# B&R Automation Studio project NAELD004C00R10L518F00 (part 10)

#### Act_OptP0410Navi.st
```iecst
ACTION Act_OptP0410Navi:

	IF tyP0410MagSel.tyNavi2Lyr1.tyBtnBack.bRtCompl = TRUE
		OR tyP0410MagSel.tyNavi2Lyr2.tyBtnBack.bRtCompl = TRUE
		OR tyP0410MagSel.tyNavi1Lyr1.tyBtnBack.bRtCompl = TRUE
		THEN
		tyP0410MagSel.tyNavi2Lyr1.tyBtnBack.bRtCompl := FALSE;
		tyP0410MagSel.tyNavi2Lyr1.tyBtnBack.bValue	:= FALSE;
		tyP0410MagSel.tyNavi2Lyr2.tyBtnBack.bRtCompl := FALSE;
		tyP0410MagSel.tyNavi2Lyr2.tyBtnBack.bValue	:= FALSE;

		tyP0410MagSel.tyNavi1Lyr1.tyBtnBack.bRtCompl := FALSE;
		tyP0410MagSel.tyNavi1Lyr1.tyBtnBack.bValue := FALSE;

		eChgPage	:= UIP0002Menu;

	ELSIF tyP0410MagSel.tyNavi2Lyr1.tyBtnLeft.bRtCompl = TRUE OR tyP0410MagSel.tyNavi2Lyr1.tyBtnRgt.bRtCompl = TRUE THEN
		tyP0410MagSel.tyNavi2Lyr1.tyBtnLeft.bRtCompl	:= FALSE;
		tyP0410MagSel.tyNavi2Lyr1.tyBtnRgt.bRtCompl	:= FALSE;

		p_tyC0004Navi ACCESS ADR(tyP0410MagSel.tyNavi2Lyr2);

		bRefreshMagRcpTable := TRUE;
		bMagazineRcpA := FALSE;
		bMagazineRcpB := TRUE;

		fUIInRtStatHide(ADR(tyP0410MagSel.tyMagDet.tyLyr.uiRtStat));

		tyP0410MagSel.tyMagSel.tyTxtMagTitle.usiValueIdx := 127;

		tyP0410MagSel.tyMagSel.tyStringRecipeNm.sValue			:= p_tyMagRcpCurrRcp1.sRcpNm;
		tyP0410MagSel.tyMagSel.tyNumMaxSlt.diValue				:= p_tyMagRcpCurrRcp1.diTtlSlt;
		tyP0410MagSel.tyMagSel.tyNumSltToSltDist.diValue		:= p_tyMagRcpCurrRcp1.diSltToSltInUM;
		tyP0410MagSel.tyMagSel.tyNumLifterMag1Slt1Pos.diValue	:= p_tyMagRcpCurrRcp1.diMag1Slt1PosInUM;
		tyP0410MagSel.tyMagSel.tyNumLifterMag2Slt1Pos.diValue	:= p_tyMagRcpCurrRcp1.diMag2Slt1PosInUM;
		tyP0410MagSel.tyMagSel.tyNumLifterMag3Slt1Pos.diValue	:= p_tyMagRcpCurrRcp1.diMag3Slt1PosInUM;
		tyP0410MagSel.tyMagSel.tyNumLifterMag4Slt1Pos.diValue	:= p_tyMagRcpCurrRcp1.diMag4Slt1PosInUM;
		tyP0410MagSel.tyMagSel.tyNumTravPosMag1.diValue			:= p_tyMagRcpCurrRcp1.diMag1TravPosInUM;
		tyP0410MagSel.tyMagSel.tyNumTravPosMag2.diValue			:= p_tyMagRcpCurrRcp1.diMag2TravPosInUM;
		tyP0410MagSel.tyMagSel.tyNumTravPosMag3.diValue			:= p_tyMagRcpCurrRcp1.diMag3TravPosInUM;
		tyP0410MagSel.tyMagSel.tyNumTravPosMag4.diValue			:= p_tyMagRcpCurrRcp1.diMag4TravPosInUM;
		tyP0410MagSel.tyMagSel.tyTxtMagModel.usiValueIdx		:= p_tyMagRcpCurrRcp1.usiMagModel;
		tyP0410MagSel.tyMagSel.tyNumMagMaxBrdWidth.diValue		:= p_tyMagRcpCurrRcp1.diMagMaxBrdWidth;
		tyP0410MagSel.tyMagSel.tyBtnSafetyBar.bValue			:= p_tyMagRcpCurrRcp1.bSafetyBarDisabled;

	ELSIF tyP0410MagSel.tyNavi2Lyr2.tyBtnLeft.bRtCompl = TRUE OR tyP0410MagSel.tyNavi2Lyr2.tyBtnRgt.bRtCompl = TRUE THEN
		tyP0410MagSel.tyNavi2Lyr2.tyBtnLeft.bRtCompl	:= FALSE;
		tyP0410MagSel.tyNavi2Lyr2.tyBtnRgt.bRtCompl	:= FALSE;

		p_tyC0004Navi ACCESS ADR(tyP0410MagSel.tyNavi2Lyr1);

		bRefreshMagRcpTable := TRUE;
		bMagazineRcpA := TRUE;
		bMagazineRcpB := FALSE;

		fUIInRtStatHide(ADR(tyP0410MagSel.tyMagDet.tyLyr.uiRtStat));

		tyP0410MagSel.tyMagSel.tyTxtMagTitle.usiValueIdx := 126;

		tyP0410MagSel.tyMagSel.tyStringRecipeNm.sValue			:= p_tyMagRcpCurrRcp.sRcpNm;
		tyP0410MagSel.tyMagSel.tyNumMaxSlt.diValue				:= p_tyMagRcpCurrRcp.diTtlSlt;
		tyP0410MagSel.tyMagSel.tyNumSltToSltDist.diValue		:= p_tyMagRcpCurrRcp.diSltToSltInUM;
		tyP0410MagSel.tyMagSel.tyNumLifterMag1Slt1Pos.diValue	:= p_tyMagRcpCurrRcp.diMag1Slt1PosInUM;
		tyP0410MagSel.tyMagSel.tyNumLifterMag2Slt1Pos.diValue	:= p_tyMagRcpCurrRcp.diMag2Slt1PosInUM;
		tyP0410MagSel.tyMagSel.tyNumLifterMag3Slt1Pos.diValue	:= p_tyMagRcpCurrRcp.diMag3Slt1PosInUM;
		tyP0410MagSel.tyMagSel.tyNumLifterMag4Slt1Pos.diValue	:= p_tyMagRcpCurrRcp.diMag4Slt1PosInUM;
		tyP0410MagSel.tyMagSel.tyNumTravPosMag1.diValue			:= p_tyMagRcpCurrRcp.diMag1TravPosInUM;
		tyP0410MagSel.tyMagSel.tyNumTravPosMag2.diValue			:= p_tyMagRcpCurrRcp.diMag2TravPosInUM;
		tyP0410MagSel.tyMagSel.tyNumTravPosMag3.diValue			:= p_tyMagRcpCurrRcp.diMag3TravPosInUM;
		tyP0410MagSel.tyMagSel.tyNumTravPosMag4.diValue			:= p_tyMagRcpCurrRcp.diMag4TravPosInUM;
		tyP0410MagSel.tyMagSel.tyTxtMagModel.usiValueIdx		:= p_tyMagRcpCurrRcp.usiMagModel;
		tyP0410MagSel.tyMagSel.tyNumMagMaxBrdWidth.diValue		:= p_tyMagRcpCurrRcp.diMagMaxBrdWidth;
		tyP0410MagSel.tyMagSel.tyBtnSafetyBar.bValue			:= p_tyMagRcpCurrRcp.bSafetyBarDisabled;
	END_IF

END_ACTION
```

#### Act_OptP0410Mask.st
```iecst
ACTION Act_OptP0410Mask:

	IF tyP0410MagSel.tyMagSel.tyBtnLoad.bRtCompl = FALSE THEN
		IF tyP0410MagSel.tyMagSel.tyTableRecipe.a_tyStringDataCol1[tyP0410Table.uiSelectedRow].sValue = '' THEN
			fUIInRtStatOff(ADR(tyP0410MagSel.tyMagSel.tyBtnLoad.uiMaskRtStat));
			fUIInRtStatOff(ADR(tyP0410MagSel.tyMagSel.tyBtnPreview.uiMaskRtStat));
		ELSE
			fUIInRtStatHide(ADR(tyP0410MagSel.tyMagSel.tyBtnLoad.uiMaskRtStat));
			fUIInRtStatHide(ADR(tyP0410MagSel.tyMagSel.tyBtnPreview.uiMaskRtStat));
		END_IF
	END_IF

	tyP0410MagSel.tyMagSel.tyBtnSort.uiMaskRtStat.0		:= (tyP0410MagSel1.tyMagSel.tyTableRecipe.a_tyStringDataCol1[1].sValue <> '') AND (tyP0410MagSel1.tyMagSel.tyBtnLoad.bRtCompl = FALSE);

END_ACTION
```

#### Act_OptP0410Load.st
```iecst
ACTION Act_OptP0410Load:

	IF tyP0410MagSel.tyMagSel.tyBtnLoad.bRtCompl = TRUE THEN

		IF usiSelMagRcpStep = 0 THEN
			//Message Confirmation Ask
			//Mask
			tyP0410MagSel.tyMagSel.tyTableRecipe.uiMaskRtStat.0		:= FALSE;
			tyP0410MagSel.tyMagSel.tyBtnPreview.uiMaskRtStat.0		:= FALSE;

			p_tyC0008MsgBox ACCESS ADR(tyP0410MagSel.tyMsgBoxSelRcpAsk);

			IF tyP0410MagSel.tyMsgBoxSelRcpAsk.tyBtnYes.bRtCompl = TRUE THEN
				tyP0410MagSel.tyMsgBoxSelRcpAsk.tyBtnYes.bRtCompl	:= FALSE;
				tyP0410MagSel.tyMsgBoxSelRcpAsk.tyBtnYes.bValue		:= FALSE;

				p_tyC0008MsgBox ACCESS ADR(tyP0410MagSel.tyMsgBoxHide);

				usiSelMagRcpStep		:= 1;

			ELSIF tyP0410MagSel.tyMsgBoxSelRcpAsk.tyBtnNo.bRtCompl = TRUE THEN
				tyP0410MagSel.tyMsgBoxSelRcpAsk.tyBtnNo.bRtCompl	:= FALSE;
				tyP0410MagSel.tyMsgBoxSelRcpAsk.tyBtnNo.bValue		:= FALSE;

				p_tyC0008MsgBox ACCESS ADR(tyP0410MagSel.tyMsgBoxHide);

				usiSelMagRcpStep		:= 99;

			END_IF

		ELSIF usiSelMagRcpStep = 1 THEN
			//Load Magazine Recipe

			IF bMagazineRcpA THEN
				tyMagRcpInfoIn.sRcpNm		:= tyP0410MagSel.tyMagSel.tyTableRecipe.a_tyStringDataCol1[tyP0410Table.uiSelectedRow].sValue;

				eMagRcpAct	:= MagRcpActLoadRcp;

				IF p_eMagRcpStat = MagRcpActLoadRcp AND p_eMagRcpStatus = Done THEN
					eMagRcpAct	:= MagRcpActIdle;

					IF p_bMagRcpNmEmpty = TRUE AND p_bMagRcpNmNotExist = TRUE THEN
						usiSelMagRcpStep	:= 2;
					ELSE

							//Update UI Current Recipe
							tyP0410MagSel.tyMagSel.tyStringRecipeNm.sValue			:= p_tyMagRcpCurrRcp.sRcpNm;
							tyP0410MagSel.tyMagSel.tyNumSltToSltDist.diValue		:= p_tyMagRcpCurrRcp.diSltToSltInUM;
							tyP0410MagSel.tyMagSel.tyNumMaxSlt.diValue				:= p_tyMagRcpCurrRcp.diTtlSlt;
							tyP0410MagSel.tyMagSel.tyNumLifterMag1Slt1Pos.diValue	:= p_tyMagRcpCurrRcp.diMag1Slt1PosInUM;
							tyP0410MagSel.tyMagSel.tyNumLifterMag2Slt1Pos.diValue	:= p_tyMagRcpCurrRcp.diMag2Slt1PosInUM;
							tyP0410MagSel.tyMagSel.tyNumLifterMag3Slt1Pos.diValue	:= p_tyMagRcpCurrRcp.diMag3Slt1PosInUM;
							tyP0410MagSel.tyMagSel.tyNumLifterMag4Slt1Pos.diValue	:= p_tyMagRcpCurrRcp.diMag4Slt1PosInUM;
							tyP0410MagSel.tyMagSel.tyNumTravPosMag1.diValue			:= p_tyMagRcpCurrRcp.diMag1TravPosInUM;
							tyP0410MagSel.tyMagSel.tyNumTravPosMag2.diValue			:= p_tyMagRcpCurrRcp.diMag2TravPosInUM;
							tyP0410MagSel.tyMagSel.tyNumTravPosMag3.diValue			:= p_tyMagRcpCurrRcp.diMag3TravPosInUM;
							tyP0410MagSel.tyMagSel.tyNumTravPosMag4.diValue			:= p_tyMagRcpCurrRcp.diMag4TravPosInUM;
							tyP0410MagSel.tyMagSel.tyTxtMagModel.usiValueIdx		:= p_tyMagRcpCurrRcp.usiMagModel;
							tyP0410MagSel.tyMagSel.tyNumMagMaxBrdWidth.diValue		:= p_tyMagRcpCurrRcp.diMagMaxBrdWidth;
							tyP0410MagSel.tyMagSel.tyBtnSafetyBar.bValue			:= p_tyMagRcpCurrRcp.bSafetyBarDisabled;
							tyP0410MagSel.tyMagSel.tyBtnMagHeightChkEn.bValue		:= p_tyMagRcpCurrRcp.bMagHeightChkEn;

							tyMagRcpCurrRcpWr	:= p_tyMagRcpCurrRcp;

							usiSelMagRcpStep	:= 99;
						END_IF

					ELSIF p_eMagRcpStatus = Error THEN
						eMagRcpAct	:= MagRcpActIdle;
						usiSelMagRcpStep		:= 99;

					END_IF

				ELSIF usiSelMagRcpStep = 2 THEN
					//Message Name Not Found
					p_tyC0008MsgBox ACCESS ADR(tyP0410MagSel.tyMsgBoxSelRcpNoNm);

					IF tyP0410MagSel.tyMsgBoxSelRcpNoNm.tyBtnNo.bRtCompl = TRUE THEN
						tyP0410MagSel.tyMsgBoxSelRcpNoNm.tyBtnNo.bRtCompl	:= FALSE;
						tyP0410MagSel.tyMsgBoxSelRcpNoNm.tyBtnNo.bValue		:= FALSE;

					p_tyC0008MsgBox ACCESS ADR(tyP0410MagSel.tyMsgBoxHide);

					usiSelMagRcpStep		:= 99;

				END_IF

			ELSIF bMagazineRcpB THEN
				tyMagRcpInfoIn1.sRcpNm		:= tyP0410MagSel.tyMagSel.tyTableRecipe.a_tyStringDataCol1[tyP0410Table.uiSelectedRow].sValue;

				eMagRcpAct1	:= MagRcpActLoadRcp;

				IF p_eMagRcpStat1 = MagRcpActLoadRcp AND p_eMagRcpStatus1 = Done THEN
					eMagRcpAct1	:= MagRcpActIdle;

					IF p_bMagRcpNmEmpty1 = TRUE AND p_bMagRcpNmNotExist1 = TRUE THEN
						usiSelMagRcpStep	:= 2;
					ELSE

						//Update UI Current Recipe
						tyP0410MagSel.tyMagSel.tyStringRecipeNm.sValue			:= p_tyMagRcpCurrRcp1.sRcpNm;
						tyP0410MagSel.tyMagSel.tyNumSltToSltDist.diValue		:= p_tyMagRcpCurrRcp1.diSltToSltInUM;
						tyP0410MagSel.tyMagSel.tyNumMaxSlt.diValue				:= p_tyMagRcpCurrRcp1.diTtlSlt;
						tyP0410MagSel.tyMagSel.tyNumLifterMag1Slt1Pos.diValue	:= p_tyMagRcpCurrRcp1.diMag1Slt1PosInUM;
						tyP0410MagSel.tyMagSel.tyNumLifterMag2Slt1Pos.diValue	:= p_tyMagRcpCurrRcp1.diMag2Slt1PosInUM;
						tyP0410MagSel.tyMagSel.tyNumLifterMag3Slt1Pos.diValue	:= p_tyMagRcpCurrRcp1.diMag3Slt1PosInUM;
						tyP0410MagSel.tyMagSel.tyNumLifterMag4Slt1Pos.diValue	:= p_tyMagRcpCurrRcp1.diMag4Slt1PosInUM;
						tyP0410MagSel.tyMagSel.tyNumTravPosMag1.diValue			:= p_tyMagRcpCurrRcp1.diMag1TravPosInUM;
						tyP0410MagSel.tyMagSel.tyNumTravPosMag2.diValue			:= p_tyMagRcpCurrRcp1.diMag2TravPosInUM;
						tyP0410MagSel.tyMagSel.tyNumTravPosMag3.diValue			:= p_tyMagRcpCurrRcp1.diMag3TravPosInUM;
						tyP0410MagSel.tyMagSel.tyNumTravPosMag4.diValue			:= p_tyMagRcpCurrRcp1.diMag4TravPosInUM;
						tyP0410MagSel.tyMagSel.tyTxtMagModel.usiValueIdx		:= p_tyMagRcpCurrRcp1.usiMagModel;
						tyP0410MagSel.tyMagSel.tyNumMagMaxBrdWidth.diValue		:= p_tyMagRcpCurrRcp1.diMagMaxBrdWidth;
						tyP0410MagSel.tyMagSel.tyBtnSafetyBar.bValue			:= p_tyMagRcpCurrRcp1.bSafetyBarDisabled;
						tyP0410MagSel.tyMagSel.tyBtnMagHeightChkEn.bValue		:= p_tyMagRcpCurrRcp1.bMagHeightChkEn;

						tyMagRcpCurrRcpWr1	:= p_tyMagRcpCurrRcp1;

						usiSelMagRcpStep	:= 99;
					END_IF

				ELSIF p_eMagRcpStatus = Error THEN
					eMagRcpAct1	:= MagRcpActIdle;
					usiSelMagRcpStep		:= 99;

				END_IF

			ELSIF usiSelMagRcpStep = 2 THEN
				//Message Name Not Found
				p_tyC0008MsgBox ACCESS ADR(tyP0410MagSel.tyMsgBoxSelRcpNoNm);

				IF tyP0410MagSel.tyMsgBoxSelRcpNoNm.tyBtnNo.bRtCompl = TRUE THEN
					tyP0410MagSel.tyMsgBoxSelRcpNoNm.tyBtnNo.bRtCompl	:= FALSE;
					tyP0410MagSel.tyMsgBoxSelRcpNoNm.tyBtnNo.bValue		:= FALSE;

					p_tyC0008MsgBox ACCESS ADR(tyP0410MagSel.tyMsgBoxHide);

					usiSelMagRcpStep		:= 99;

				END_IF
			END_IF

		ELSIF usiSelMagRcpStep = 99 THEN
			//Complete
			//Unmask
			tyP0410MagSel.tyMagSel.tyTableRecipe.uiMaskRtStat.0		:= TRUE;
			tyP0410MagSel.tyMagSel.tyBtnPreview.uiMaskRtStat.0		:= TRUE;

			//Reset
			tyP0410MagSel.tyMagSel.tyBtnLoad.bRtCompl				:= FALSE;
			tyP0410MagSel.tyMagSel.tyBtnLoad.bValue					:= FALSE;

			usiSelMagRcpStep			:= 0;

		END_IF

	END_IF

END_ACTION
```

#### Act_OptP0410Preview.st
```iecst
ACTION Act_OptP0410Preview:

	IF tyP0410MagSel.tyMagSel.tyBtnPreview.bRtCompl = TRUE THEN
		IF bMagazineRcpA THEN
			tyMagRcpInfoIn.sRcpNm	:= tyP0410MagSel.tyMagSel.tyTableRecipe.a_tyStringDataCol1[tyP0410Table.uiSelectedRow].sValue;

			eMagRcpAct				:= MagRcpActGetInfo;

			IF	p_eMagRcpStat = MagRcpActGetInfo AND p_eMagRcpStatus = Done THEN
				eMagRcpAct			:= MagRcpActIdle;

				IF p_bMagRcpNmEmpty = TRUE AND p_bMagRcpNmNotExist = TRUE THEN

					tyP0410MagSel.tyMagDet.tyStringRecipeNm.sValue			:= '';
					tyP0410MagSel.tyMagDet.tyNumSltToSltDist.diValue		:= 0;
					tyP0410MagSel.tyMagDet.tyNumMaxSlt.diValue				:= 0;
					tyP0410MagSel.tyMagDet.tyNumLifterMag1Slt1Pos.diValue	:= 0;
					tyP0410MagSel.tyMagDet.tyNumLifterMag2Slt1Pos.diValue	:= 0;
					tyP0410MagSel.tyMagDet.tyNumLifterMag3Slt1Pos.diValue	:= 0;
					tyP0410MagSel.tyMagDet.tyNumLifterMag4Slt1Pos.diValue	:= 0;
					tyP0410MagSel.tyMagDet.tyNumTravPosMag1.diValue			:= 0;
					tyP0410MagSel.tyMagDet.tyNumTravPosMag2.diValue			:= 0;
					tyP0410MagSel.tyMagDet.tyNumTravPosMag3.diValue			:= 0;
					tyP0410MagSel.tyMagDet.tyNumTravPosMag4.diValue			:= 0;
					tyP0410MagSel.tyMagDet.tyNumMagMaxBrdWidth.diValue		:= 0;
					tyP0410MagSel.tyMagDet.tyBtnSafetyBar.bValue			:= FALSE;
					tyP0410MagSel.tyMagDet.tyBtnMagHeightChkEn.bValue		:= FALSE;

				ELSE

					tyP0410MagSel.tyMagDet.tyStringRecipeNm.sValue			:= p_tyMagRcpInfoOut.sRcpNm;
					tyP0410MagSel.tyMagDet.tyNumSltToSltDist.diValue		:= p_tyMagRcpInfoOut.diSltToSltInUM;
					tyP0410MagSel.tyMagDet.tyNumMaxSlt.diValue				:= p_tyMagRcpInfoOut.diTtlSlt;
					tyP0410MagSel.tyMagDet.tyNumLifterMag1Slt1Pos.diValue	:= p_tyMagRcpInfoOut.diMag1Slt1PosInUM;
					tyP0410MagSel.tyMagDet.tyNumLifterMag2Slt1Pos.diValue	:= p_tyMagRcpInfoOut.diMag2Slt1PosInUM;
					tyP0410MagSel.tyMagDet.tyNumLifterMag3Slt1Pos.diValue	:= p_tyMagRcpInfoOut.diMag3Slt1PosInUM;
					tyP0410MagSel.tyMagDet.tyNumLifterMag4Slt1Pos.diValue	:= p_tyMagRcpInfoOut.diMag4Slt1PosInUM;
					tyP0410MagSel.tyMagDet.tyNumTravPosMag1.diValue			:= p_tyMagRcpInfoOut.diMag1TravPosInUM;
					tyP0410MagSel.tyMagDet.tyNumTravPosMag2.diValue			:= p_tyMagRcpInfoOut.diMag2TravPosInUM;
					tyP0410MagSel.tyMagDet.tyNumTravPosMag3.diValue			:= p_tyMagRcpInfoOut.diMag3TravPosInUM;
					tyP0410MagSel.tyMagDet.tyNumTravPosMag4.diValue			:= p_tyMagRcpInfoOut.diMag4TravPosInUM;
					tyP0410MagSel.tyMagDet.tyNumMagMaxBrdWidth.diValue		:= p_tyMagRcpInfoOut.diMagMaxBrdWidth;
					tyP0410MagSel.tyMagDet.tyBtnSafetyBar.bValue			:= p_tyMagRcpInfoOut.bSafetyBarDisabled;
					tyP0410MagSel.tyMagDet.tyBtnMagHeightChkEn.bValue		:= p_tyMagRcpInfoOut.bMagHeightChkEn;
				END_IF

				fUIInRtStatOff(ADR(tyP0410MagSel.tyMagDet.tyLyr.uiRtStat));

				tyP0410MagSel.tyMagSel.tyBtnPreview.bRtCompl				:= FALSE;
			END_IF

		ELSIF bMagazineRcpB THEN

			tyMagRcpInfoIn1.sRcpNm	:= tyP0410MagSel.tyMagSel.tyTableRecipe.a_tyStringDataCol1[tyP0410Table.uiSelectedRow].sValue;

			eMagRcpAct1				:= MagRcpActGetInfo;

			IF	p_eMagRcpStat1 = MagRcpActGetInfo AND p_eMagRcpStatus1 = Done THEN
				eMagRcpAct1			:= MagRcpActIdle;

				IF p_bMagRcpNmEmpty1 = TRUE AND p_bMagRcpNmNotExist1 = TRUE THEN

					tyP0410MagSel.tyMagDet.tyStringRecipeNm.sValue			:= '';
					tyP0410MagSel.tyMagDet.tyNumSltToSltDist.diValue		:= 0;
					tyP0410MagSel.tyMagDet.tyNumMaxSlt.diValue				:= 0;
					tyP0410MagSel.tyMagDet.tyNumLifterMag1Slt1Pos.diValue	:= 0;
					tyP0410MagSel.tyMagDet.tyNumLifterMag2Slt1Pos.diValue	:= 0;
					tyP0410MagSel.tyMagDet.tyNumLifterMag3Slt1Pos.diValue	:= 0;
					tyP0410MagSel.tyMagDet.tyNumLifterMag4Slt1Pos.diValue	:= 0;
					tyP0410MagSel.tyMagDet.tyNumTravPosMag1.diValue			:= 0;
					tyP0410MagSel.tyMagDet.tyNumTravPosMag2.diValue			:= 0;
					tyP0410MagSel.tyMagDet.tyNumTravPosMag3.diValue			:= 0;
					tyP0410MagSel.tyMagDet.tyNumTravPosMag4.diValue			:= 0;
					tyP0410MagSel.tyMagDet.tyNumMagMaxBrdWidth.diValue		:= 0;
					tyP0410MagSel.tyMagDet.tyBtnSafetyBar.bValue			:= FALSE;
					tyP0410MagSel.tyMagDet.tyBtnMagHeightChkEn.bValue		:= FALSE;
				ELSE

					tyP0410MagSel.tyMagDet.tyStringRecipeNm.sValue			:= p_tyMagRcpInfoOut1.sRcpNm;
					tyP0410MagSel.tyMagDet.tyNumSltToSltDist.diValue		:= p_tyMagRcpInfoOut1.diSltToSltInUM;
					tyP0410MagSel.tyMagDet.tyNumMaxSlt.diValue				:= p_tyMagRcpInfoOut1.diTtlSlt;
					tyP0410MagSel.tyMagDet.tyNumLifterMag1Slt1Pos.diValue	:= p_tyMagRcpInfoOut1.diMag1Slt1PosInUM;
					tyP0410MagSel.tyMagDet.tyNumLifterMag2Slt1Pos.diValue	:= p_tyMagRcpInfoOut1.diMag2Slt1PosInUM;
					tyP0410MagSel.tyMagDet.tyNumLifterMag3Slt1Pos.diValue	:= p_tyMagRcpInfoOut1.diMag3Slt1PosInUM;
					tyP0410MagSel.tyMagDet.tyNumLifterMag4Slt1Pos.diValue	:= p_tyMagRcpInfoOut1.diMag4Slt1PosInUM;
					tyP0410MagSel.tyMagDet.tyNumTravPosMag1.diValue			:= p_tyMagRcpInfoOut1.diMag1TravPosInUM;
					tyP0410MagSel.tyMagDet.tyNumTravPosMag2.diValue			:= p_tyMagRcpInfoOut1.diMag2TravPosInUM;
					tyP0410MagSel.tyMagDet.tyNumTravPosMag3.diValue			:= p_tyMagRcpInfoOut1.diMag3TravPosInUM;
					tyP0410MagSel.tyMagDet.tyNumTravPosMag4.diValue			:= p_tyMagRcpInfoOut1.diMag4TravPosInUM;
					tyP0410MagSel.tyMagDet.tyNumMagMaxBrdWidth.diValue		:= p_tyMagRcpInfoOut1.diMagMaxBrdWidth;
					tyP0410MagSel.tyMagDet.tyBtnSafetyBar.bValue			:= p_tyMagRcpInfoOut1.bSafetyBarDisabled;
					tyP0410MagSel.tyMagDet.tyBtnMagHeightChkEn.bValue		:= p_tyMagRcpInfoOut1.bMagHeightChkEn;
				END_IF

				fUIInRtStatOff(ADR(tyP0410MagSel.tyMagDet.tyLyr.uiRtStat));

				tyP0410MagSel.tyMagSel.tyBtnPreview.bRtCompl				:= FALSE;
			END_IF
		END_IF
	END_IF

	IF tyP0410MagSel.tyMagDet.tyHotspotClose.bRtCompl = TRUE THEN
		tyP0410MagSel.tyMagDet.tyHotspotClose.bRtCompl					:= FALSE;
		tyP0410MagSel.tyMagSel.tyBtnPreview.bValue						:= FALSE;

		//Hide Recipe Details
		fUIInRtStatHide(ADR(tyP0410MagSel.tyMagDet.tyLyr.uiRtStat));
	END_IF

END_ACTION
```

#### Act_OptP0410Table.st
```iecst
ACTION Act_OptP0410Table:

	//Call Table FB
	fbP0410Table.sVisuNm			:= tyP0410Table.sVisuNm;
	fbP0410Table.udiWorkAreaStartX	:= 349;
	fbP0410Table.udiWorkAreaEndX	:= 768;
	fbP0410Table.udiWorkAreaStartY	:= 107;
	fbP0410Table.udiWorkAreaEndY	:= 428;
	fbP0410Table.udiMinXDist		:= 20;
	fbP0410Table.udiMinYDist		:= 20;
	fbP0410Table.uiSlideScale		:= c_uiP0410TableSize;
	fbP0410Table.iTotalData			:= UDINT_TO_INT(c_udiMagRcpMax);;
	fbP0410Table.iTotalRow			:= c_uiP0410TableSize;
	fbP0410Table(uiSliderStatus := tyP0410MagSel.tyMagSel.tyTableRecipe.tyUISlider.uiRtStat , a_tyUIHotspot := tyP0410MagSel.tyMagSel.tyTableRecipe.a_tyHotspot , uiTablePos := tyP0410Table.uiTablePos , iSliderPos := tyP0410MagSel.tyMagSel.tyTableRecipe.tyUISlider.iValue);

	tyP0410Table.uiSelectedRow		:= fbP0410Table.uiSelectedRow;
	tyP0410Table.bTableActive		:= fbP0410Table.bTableActive;
	tyP0410Table.bSliderActive		:= fbP0410Table.bSliderActive;

	//Table Content
	IF tyP0410Table.bTableActive = TRUE OR tyP0410Table.bSliderActive = TRUE OR bRefreshMagRcpTable OR bUpdateP0410Table THEN

		IF bMagazineRcpA THEN
			FOR i := 1 TO c_uiP0410TableSize DO

				IF tyP0410MagSel.tyMagSel.tyBtnSort.bValue THEN

					tyP0410MagSel.tyMagSel.tyTableRecipe.a_tyStringDataCol0[i].sValue	:= UINT_TO_STRING(tyP0410Table.uiTablePos + i - 1);
					tyP0410MagSel.tyMagSel.tyTableRecipe.a_tyStringDataCol1[i].sValue	:= p_tyMagRcpSortedList[tyP0410Table.uiTablePos + i - 1].sRcpNm;
					tyP0410MagSel.tyMagSel.tyTableRecipe.a_tyStringDataCol2[i].sValue	:= p_tyMagRcpSortedList[tyP0410Table.uiTablePos + i - 1].sDisplayInfo;

				ELSE
					tyP0410MagSel.tyMagSel.tyTableRecipe.a_tyStringDataCol0[i].sValue	    := UINT_TO_STRING(tyP0410Table.uiTablePos + i - 1);
					tyP0410MagSel.tyMagSel.tyTableRecipe.a_tyStringDataCol1[i].sValue		:= p_tyMagRcpCurrList[tyP0410Table.uiTablePos + i - 1].sRcpNm;
					tyP0410MagSel.tyMagSel.tyTableRecipe.a_tyStringDataCol2[i].sValue		:= p_tyMagRcpCurrList[tyP0410Table.uiTablePos + i - 1].sDisplayInfo;
				END_IF

			END_FOR

		ELSIF bMagazineRcpB THEN
			FOR i := 1 TO c_uiP0410TableSize DO

				IF tyP0410MagSel.tyMagSel.tyBtnSort.bValue THEN

					tyP0410MagSel.tyMagSel.tyTableRecipe.a_tyStringDataCol0[i].sValue	:= UINT_TO_STRING(tyP0410Table.uiTablePos + i - 1);
					tyP0410MagSel.tyMagSel.tyTableRecipe.a_tyStringDataCol1[i].sValue	:= p_tyMagRcpSortedList1[tyP0410Table.uiTablePos + i - 1].sRcpNm;
					tyP0410MagSel.tyMagSel.tyTableRecipe.a_tyStringDataCol2[i].sValue	:= p_tyMagRcpSortedList1[tyP0410Table.uiTablePos + i - 1].sDisplayInfo;

				ELSE
					tyP0410MagSel.tyMagSel.tyTableRecipe.a_tyStringDataCol0[i].sValue	    := UINT_TO_STRING(tyP0410Table.uiTablePos + i - 1);
					tyP0410MagSel.tyMagSel.tyTableRecipe.a_tyStringDataCol1[i].sValue		:= p_tyMagRcpCurrList1[tyP0410Table.uiTablePos + i - 1].sRcpNm;
					tyP0410MagSel.tyMagSel.tyTableRecipe.a_tyStringDataCol2[i].sValue		:= p_tyMagRcpCurrList1[tyP0410Table.uiTablePos + i - 1].sDisplayInfo;
				END_IF

			END_FOR
		END_IF

		IF bUpdateP0410Table THEN
			bUpdateP0410Table := FALSE;
		END_IF
	END_IF

	//Selected Row
	IF tyP0410Table.uiSelectedRow <> tyP0410Table.uiSelectedRowOld THEN
		FOR i := 1 TO c_uiP0410TableSize DO
			IF tyP0410Table.uiSelectedRow = i THEN
				tyP0410MagSel.tyMagSel.tyTableRecipe.a_tyStringDataCol1[i].usiColor	:= 1;
				tyP0410MagSel.tyMagSel.tyTableRecipe.a_tyStringDataCol2[i].usiColor	:= 1;
			ELSE
				tyP0410MagSel.tyMagSel.tyTableRecipe.a_tyStringDataCol1[i].usiColor	:= 0;
				tyP0410MagSel.tyMagSel.tyTableRecipe.a_tyStringDataCol2[i].usiColor	:= 0;
			END_IF

			//Magazine B
			IF tyP0410Table.uiSelectedRow = i THEN
				tyP0410MagSel1.tyMagSel.tyTableRecipe.a_tyStringDataCol1[i].usiColor	:= 1;
				tyP0410MagSel1.tyMagSel.tyTableRecipe.a_tyStringDataCol2[i].usiColor	:= 1;
			ELSE
				tyP0410MagSel1.tyMagSel.tyTableRecipe.a_tyStringDataCol1[i].usiColor	:= 0;
				tyP0410MagSel1.tyMagSel.tyTableRecipe.a_tyStringDataCol2[i].usiColor	:= 0;
			END_IF
		END_FOR

		tyP0410Table.uiSelectedRowOld	:= tyP0410Table.uiSelectedRow;
	END_IF

END_ACTION
```

#### Act_OptP0410Sort.st
```iecst
ACTION Act_OptP0410Sort:

	IF tyP0410MagSel.tyMagSel.tyBtnSort.bValue THEN
		tyP0410MagSel.tyMagSel.tyBtnSort.usiTxtIdx 	:= 1;
	ELSE
		tyP0410MagSel.tyMagSel.tyBtnSort.usiTxtIdx 	:= 0;
	END_IF

	IF tyP0410MagSel.tyMagSel.tyBtnSort.bRtCompl THEN

		IF tyP0410MagSel.tyMagSel.tyBtnSort.bValue THEN

			tyP0410MagSel.tyMagSel.tyTableRecipe.uiMaskRtStat.0	:= FALSE;

			eMagRcpAct	:= MagRcpActSort;
			eMagRcpAct1	:= MagRcpActSort;
			IF p_eMagRcpStat = MagRcpActSort AND p_eMagRcpStatus = Done
				AND (p_eMagRcpStat1 = MagRcpActSort AND p_eMagRcpStatus1 = Done)
				THEN
				eMagRcpAct		:= MagRcpActIdle;
				eMagRcpAct1		:= MagRcpActIdle;
				FOR i := 1 TO c_uiP0410TableSize DO
					tyP0410MagSel.tyMagSel.tyTableRecipe.a_tyStringDataCol0[i].sValue	:= UINT_TO_STRING(tyP0400Table.uiTablePos + i - 1);
					tyP0410MagSel.tyMagSel.tyTableRecipe.a_tyStringDataCol1[i].sValue	:= p_tyMagRcpSortedList[tyP0400Table.uiTablePos + i - 1].sRcpNm;
					tyP0410MagSel.tyMagSel.tyTableRecipe.a_tyStringDataCol2[i].sValue	:= p_tyMagRcpSortedList[tyP0400Table.uiTablePos + i - 1].sDisplayInfo;
				END_FOR

				//Unmask
				tyP0410MagSel.tyMagSel.tyTableRecipe.uiMaskRtStat.0	:= TRUE;

				tyP0410MagSel.tyMagSel.tyBtnSort.bRtCompl := FALSE;

			ELSIF p_eMagRcpStatus = Error OR p_eMagRcpStatus1 = Error THEN
				FOR i := 1 TO c_uiP0410TableSize DO
					tyP0410MagSel.tyMagSel.tyTableRecipe.a_tyStringDataCol0[i].sValue		:= UINT_TO_STRING(tyP0410Table.uiTablePos + i - 1);
					tyP0410MagSel.tyMagSel.tyTableRecipe.a_tyStringDataCol1[i].sValue		:= '';
					tyP0410MagSel.tyMagSel.tyTableRecipe.a_tyStringDataCol2[i].sValue		:= '';
				END_FOR
				eMagRcpAct		:= MagRcpActIdle;
				eMagRcpAct1		:= MagRcpActIdle;
				p_tyC0008MsgBox ACCESS ADR (tyP0410MagSel.tyMsgBoxListErr);

				IF tyP0410MagSel.tyMsgBoxListErr.tyBtnNo.bRtCompl = TRUE THEN
					tyP0410MagSel.tyMsgBoxListErr.tyBtnNo.bRtCompl 		:= TRUE;
					tyP0410MagSel.tyMsgBoxListErr.tyBtnNo.bValue			:= TRUE;

					p_tyC0008MsgBox ACCESS ADR (tyP0410MagSel.tyMsgBoxHide);

					//Unmask
					tyP0410MagSel.tyMagSel.tyTableRecipe.uiMaskRtStat.0	:= TRUE;

					//Reset
					tyP0410MagSel.tyMagSel.tyBtnSort.bRtCompl := FALSE;
				END_IF
			END_IF

		ELSE

			bUpdateP0410Table	:= TRUE;

			tyP0410MagSel.tyMagSel.tyBtnSort.bRtCompl := FALSE;

		END_IF

	END_IF

END_ACTION
```

#### Act_EntP0600Disp.st
```iecst
ACTION Act_EntP0600Disp:

	//Access Addres
	p_tyC0005Main ACCESS ADR(tyCommon.tyMain);

	p_tyC0007Notif ACCESS ADR(tyCommon.tyNotif);

	p_tyC0008MsgBox ACCESS ADR(tyP0600Alm.tyMsgBoxHide);

	p_tyC0009Info ACCESS ADR(tyCommon.tyInfo);

	p_tyC0010RcyMsg ACCESS ADR(tyP0600Alm.tyRcyMsgHide);

	p_tyP0600Alm ACCESS ADR(tyP0600Alm.tyAlm);

	tyP0600Alm.tyAlm.tyBtnCurr.bRtCompl := TRUE; //Default will be Current Alarm View

	//Reset
	bTeachTravPosA			:= FALSE;
	bTeachTravPosB			:= FALSE;
	bTeachLifterPosA		:= FALSE;
	bTeachLifterPosB		:= FALSE;
	bTeachLifterMag1Slt1Pos	:= FALSE;
	bTeachLifterMag2Slt1Pos	:= FALSE;
	bTeachLifterMag3Slt1Pos	:= FALSE;
	bTeachLifterMag4Slt1Pos	:= FALSE;
	bTeachTravPosMag1		:= FALSE;
	bTeachTravPosMag2		:= FALSE;
	bTeachTravPosMag3		:= FALSE;
	bTeachTravPosMag4		:= FALSE;
	bTeachServo				:= FALSE;

END_ACTION
```

#### Act_OptP0600Alm.st
```iecst
ACTION Act_OptP0600Alm:

	IF tyP0600Alm.tyAlm.tyBtnHistory.bRtCompl = TRUE THEN
		tyP0600Alm.tyAlm.tyBtnHistory.bRtCompl		:= FALSE;
		tyP0600Alm.tyAlm.tyBtnHistory.bValue		:= TRUE;
		tyP0600Alm.tyAlm.tyBtnCurr.bValue			:= FALSE;
	ELSIF tyP0600Alm.tyAlm.tyBtnCurr.bRtCompl = TRUE THEN
		tyP0600Alm.tyAlm.tyBtnCurr.bRtCompl			:= FALSE;
		tyP0600Alm.tyAlm.tyBtnCurr.bValue			:= TRUE;
		tyP0600Alm.tyAlm.tyBtnHistory.bValue		:= FALSE;
	END_IF

	IF NOT p_bAlarmErr THEN
		memset(ADR(tyUIAlmData.bAlm) , 0 , SIZEOF(tyUIAlmData.bAlm));
	END_IF

	IF NOT p_bAlarmWarning THEN
		memset(ADR(tyUIAlmData.bWarning) , 0 , SIZEOF(tyUIAlmData.bWarning));
	ELSE
		IF p_bDSHermesAConnected OR p_tyMcParamCurr.eDSCommA = McSetCommModSMEMA THEN
			tyUIAlmData.bWarning[3363] := FALSE;
		END_IF
		IF p_bDSHermesBConnected OR p_tyMcParamCurr.eDSCommB = McSetCommModSMEMA THEN
			tyUIAlmData.bWarning[3531] := FALSE;
		END_IF
	END_IF

	IF tyP0600Alm.tyAlm.tyBtnCurr.bValue = TRUE THEN

		fUIInRtStatOff(ADR(tyP0600Alm.tyAlm.tyAlarm.tyUIAlmCur.uiRtStat));
		fUIInRtStatHide(ADR(tyP0600Alm.tyAlm.tyAlarm.tyUIAlmHis.uiRtStat));
		tyP0600Alm.tyAlm.tyBtnHistoryUp.uiMaskRtStat.0 		:= FALSE;
		tyP0600Alm.tyAlm.tyBtnHistoryDown.uiMaskRtStat.0 	:= FALSE;

		FOR i := 1 TO c_uiP0600TableSize DO
			IF p_bStartupUISettingsLoadDone THEN
				IF p_tyAlarmCurrList[i].eSeverity = AlmSeverityError THEN
					tyUIAlmData.bAlm[p_tyAlarmCurrList[i].udiErrorCode] := p_tyAlarmCurrList[i].bAlm;
				ELSIF p_tyAlarmCurrList[i].eSeverity = AlmSeverityWarning THEN
					tyUIAlmData.bWarning[p_tyAlarmCurrList[i].udiErrorCode] := p_tyAlarmCurrList[i].bWarning;
				END_IF
			END_IF
		END_FOR

	ELSIF tyP0600Alm.tyAlm.tyBtnHistory.bValue = TRUE THEN

		fUIInRtStatHide(ADR(tyP0600Alm.tyAlm.tyAlarm.tyUIAlmCur.uiRtStat));
		fUIInRtStatOff(ADR(tyP0600Alm.tyAlm.tyAlarm.tyUIAlmHis.uiRtStat));
		tyP0600Alm.tyAlm.tyBtnHistoryUp.uiMaskRtStat.0 		:= TRUE;
		tyP0600Alm.tyAlm.tyBtnHistoryDown.uiMaskRtStat.0 	:= TRUE;

	END_IF

END_ACTION
```

#### Act_OptP0700Table.st
```iecst
ACTION Act_OptP0700Table:

	//Call Table FB
	fbP0700Table.sVisuNm			:= tyP0700Table.sVisuNm;
	fbP0700Table.udiWorkAreaStartX	:= 17;
	fbP0700Table.udiWorkAreaEndX	:= 594;
	fbP0700Table.udiWorkAreaStartY	:= 94;
	fbP0700Table.udiWorkAreaEndY	:= 445;
	fbP0700Table.udiMinXDist		:= 20;
	fbP0700Table.udiMinYDist		:= 20;
	fbP0700Table.uiSlideScale		:= c_uiP0700TableSize;
	fbP0700Table.iTotalData			:= UDINT_TO_INT(c_diLFClntNum);
	fbP0700Table.iTotalRow			:= c_uiP0700TableSize;
	fbP0700Table(uiSliderStatus 	:= tyP0700LFCtrl.tyLdr.tyTable1List.tyUISlider.uiRtStat , a_tyUIHotspot := tyP0700LFCtrl.tyLdr.tyTable1List.a_tyHotspot , uiTablePos := tyP0700Table.uiTablePos , iSliderPos := tyP0700LFCtrl.tyLdr.tyTable1List.tyUISlider.iValue);

	tyP0700Table.uiSelectedRow		:= fbP0700Table.uiSelectedRow;
	tyP0700Table.bTableActive		:= fbP0700Table.bTableActive;
	tyP0700Table.bSliderActive		:= fbP0700Table.bSliderActive;

	//Table Content
	IF tyP0700Table.bTableActive = TRUE OR tyP0700Table.bSliderActive = TRUE THEN
		FOR i := 1 TO c_uiP0700TableSize DO
			tyP0700LFCtrl.tyLdr.tyTable1List.a_tyStringDataCol0[i].sValue	:= UINT_TO_STRING(tyP0700Table.uiTablePos + i - 1);
		END_FOR
	END_IF

	//Update Status & Current Recipe
	FOR i := 1 TO c_uiP0700TableSize DO
		tyP0700LFCtrl.tyLdr.tyTable1List.a_tyStringDataCol1[i].sValue	:= p_tyLFLeaderFollowerToLeaderTag[tyP0700Table.uiTablePos + i - 1].sMcNm;
		tyP0700LFCtrl.tyLdr.tyTable1List.a_tyStringDataCol2[i].sValue	:= p_tyMcParamCurr.a_sLFIPAddr[tyP0700Table.uiTablePos + i - 1];
		tyP0700LFCtrl.tyLdr.tyTable1List.a_tyStringDataCol4[i].sValue	:= p_tyLFLeaderFollowerToLeaderTag[tyP0700Table.uiTablePos + i - 1].sCurrProdRcp;

		IF p_tyMcParamCurr.a_sLFIPAddr[tyP0700Table.uiTablePos + i - 1] = '' THEN
			tyP0700LFCtrl.tyLdr.tyTable1List.a_tyTxtDataCol3[i].usiValueIdx	:= 0;	//Empty
		ELSIF p_tyMcParamCurr.a_sLFIPAddr[tyP0700Table.uiTablePos + i - 1] = '0000' THEN
			tyP0700LFCtrl.tyLdr.tyTable1List.a_tyTxtDataCol3[i].usiValueIdx	:= 3;	//Third Party
		ELSIF p_tyMcParamCurr.a_bLFOnline[tyP0700Table.uiTablePos + i - 1] = FALSE THEN
			tyP0700LFCtrl.tyLdr.tyTable1List.a_tyTxtDataCol3[i].usiValueIdx	:= 9;	//Offline
		ELSIF p_tyMcParamCurr.a_sLFIPAddr[tyP0700Table.uiTablePos + i - 1] = p_sHWInfoIPAddr THEN
			tyP0700LFCtrl.tyLdr.tyTable1List.a_tyTxtDataCol3[i].usiValueIdx	:= 4;	//Leader
		ELSIF p_tyLFLeaderFollowerToLeaderTag[tyP0700Table.uiTablePos + i - 1].bSectionLeader = TRUE THEN
			tyP0700LFCtrl.tyLdr.tyTable1List.a_tyTxtDataCol3[i].usiValueIdx	:= 5;	//Section Leader
		ELSIF p_tyLFLeaderFollowerInfo[tyP0700Table.uiTablePos + i - 1].bOnline = FALSE THEN
			tyP0700LFCtrl.tyLdr.tyTable1List.a_tyTxtDataCol3[i].usiValueIdx	:= 9;	//Offline
		ELSE
			IF p_tyLFLeaderFollowerToLeaderTag[tyP0700Table.uiTablePos + i - 1].eCurrMachineStat=Run THEN
				IF p_tyLFLeaderFollowerToLeaderTag[tyP0700Table.uiTablePos + i - 1].eCurrMachineStat=Warning THEN
					tyP0700LFCtrl.tyLdr.tyTable1List.a_tyTxtDataCol3[i].usiValueIdx	:= 2;	//Warning
				ELSE
					tyP0700LFCtrl.tyLdr.tyTable1List.a_tyTxtDataCol3[i].usiValueIdx	:= 6;	//Run
				END_IF
			ELSE
				IF p_tyLFLeaderFollowerToLeaderTag[tyP0700Table.uiTablePos + i - 1].eCurrMachineStat=InError THEN
					tyP0700LFCtrl.tyLdr.tyTable1List.a_tyTxtDataCol3[i].usiValueIdx	:= 1;	//Error
				ELSIF p_tyLFLeaderFollowerToLeaderTag[tyP0700Table.uiTablePos + i - 1].eCurrMachineStat=Warning THEN
					tyP0700LFCtrl.tyLdr.tyTable1List.a_tyTxtDataCol3[i].usiValueIdx	:= 2;	//Warning
				ELSIF p_tyLFLeaderFollowerToLeaderTag[tyP0700Table.uiTablePos + i - 1].eCurrMachineStat=Manual THEN
					tyP0700LFCtrl.tyLdr.tyTable1List.a_tyTxtDataCol3[i].usiValueIdx	:= 8;	//Manual
				ELSE
					tyP0700LFCtrl.tyLdr.tyTable1List.a_tyTxtDataCol3[i].usiValueIdx	:= 7;	//Stop
				END_IF
			END_IF
		END_IF
	END_FOR

	//Update Color
	FOR i := 1 TO c_uiP0700TableSize DO

		IF p_tyMcParamCurr.a_sLFIPAddr[tyP0700Table.uiTablePos + i - 1] = '' THEN
			tyP0700LFCtrl.tyLdr.tyTable1List.a_tyTxtDataCol3[i].usiColor	:= 0;	//Empty
		ELSIF p_tyMcParamCurr.a_sLFIPAddr[tyP0700Table.uiTablePos + i - 1] = '0000' THEN
			tyP0700LFCtrl.tyLdr.tyTable1List.a_tyTxtDataCol3[i].usiColor	:= 0;	//Third Party
		ELSIF p_tyMcParamCurr.a_bLFOnline[tyP0700Table.uiTablePos + i - 1] = FALSE THEN
			tyP0700LFCtrl.tyLdr.tyTable1List.a_tyTxtDataCol3[i].usiColor	:= 3;	//Offline
		ELSIF p_tyMcParamCurr.a_sLFIPAddr[tyP0700Table.uiTablePos + i - 1] = p_sHWInfoIPAddr THEN
			IF p_bOpsRun THEN
				tyP0700LFCtrl.tyLdr.tyTable1List.a_tyTxtDataCol3[i].usiColor	:= 1;	//Leader Run
			ELSE
				tyP0700LFCtrl.tyLdr.tyTable1List.a_tyTxtDataCol3[i].usiColor	:= 2;	//Leader Stop
			END_IF
		ELSIF p_tyLFLeaderFollowerToLeaderTag[tyP0700Table.uiTablePos + i - 1].bSectionLeader = TRUE THEN
			IF p_tyLFLeaderFollowerToLeaderTag[tyP0700Table.uiTablePos + i - 1].eCurrMachineStat=Run THEN
				tyP0700LFCtrl.tyLdr.tyTable1List.a_tyTxtDataCol3[i].usiColor	:= 1;	//Section Leader Run
			ELSE
				tyP0700LFCtrl.tyLdr.tyTable1List.a_tyTxtDataCol3[i].usiColor	:= 2;	//Section Leader Stop
			END_IF
		ELSIF p_tyLFLeaderFollowerInfo[tyP0700Table.uiTablePos + i - 1].bOnline = FALSE THEN
			tyP0700LFCtrl.tyLdr.tyTable1List.a_tyTxtDataCol3[i].usiColor	:= 3;	//Offline
		ELSE
			IF p_tyLFLeaderFollowerToLeaderTag[tyP0700Table.uiTablePos + i - 1].eCurrMachineStat=Run THEN
				IF p_tyLFLeaderFollowerToLeaderTag[tyP0700Table.uiTablePos + i - 1].eCurrMachineStat=Warning THEN
					tyP0700LFCtrl.tyLdr.tyTable1List.a_tyTxtDataCol3[i].usiColor	:= 4;	//Warning
				ELSE
					tyP0700LFCtrl.tyLdr.tyTable1List.a_tyTxtDataCol3[i].usiColor	:= 1;	//Run
				END_IF
			ELSE
				IF p_tyLFLeaderFollowerToLeaderTag[tyP0700Table.uiTablePos + i - 1].eCurrMachineStat=InError THEN
					tyP0700LFCtrl.tyLdr.tyTable1List.a_tyTxtDataCol3[i].usiColor	:= 2;	//Error
				ELSIF p_tyLFLeaderFollowerToLeaderTag[tyP0700Table.uiTablePos + i - 1].eCurrMachineStat=Warning THEN
					tyP0700LFCtrl.tyLdr.tyTable1List.a_tyTxtDataCol3[i].usiColor	:= 4;	//Warning
				ELSIF p_tyLFLeaderFollowerToLeaderTag[tyP0700Table.uiTablePos + i - 1].eCurrMachineStat=Manual THEN
					tyP0700LFCtrl.tyLdr.tyTable1List.a_tyTxtDataCol3[i].usiColor	:= 6;	//Manual
				ELSE
					tyP0700LFCtrl.tyLdr.tyTable1List.a_tyTxtDataCol3[i].usiColor	:= 5;	//Stop
				END_IF
			END_IF
		END_IF

	END_FOR

END_ACTION
```

#### Act_EntP0800Disp.st
```iecst
ACTION Act_EntP0800Disp:

	//Access Address
	IF p_tyNtParamCurr.eProjMag = LDMagQuadruple THEN
		IF bDisplayMag4Info THEN
			p_tyC0004Navi ACCESS ADR(tyP0800MagInfo.tyNaviLyr2);

			fUIInRtStatHide(ADR(tyP0800MagInfo.tyMagInfo1.tyLyr.uiRtStat));
			fUIInRtStatHide(ADR(tyP0800MagInfo.tyMagInfo2.tyLyr.uiRtStat));
			fUIInRtStatHide(ADR(tyP0800MagInfo.tyMagInfo3.tyLyr.uiRtStat));
			fUIInRtStatOff(ADR(tyP0800MagInfo.tyMagInfo4.tyLyr.uiRtStat));

		ELSE

			p_tyC0004Navi ACCESS ADR(tyP0800MagInfo.tyNaviLyr1);

			fUIInRtStatOff(ADR(tyP0800MagInfo.tyMagInfo1.tyLyr.uiRtStat));
			fUIInRtStatOff(ADR(tyP0800MagInfo.tyMagInfo2.tyLyr.uiRtStat));
			fUIInRtStatOff(ADR(tyP0800MagInfo.tyMagInfo3.tyLyr.uiRtStat));
			fUIInRtStatHide(ADR(tyP0800MagInfo.tyMagInfo4.tyLyr.uiRtStat));

		END_IF
	ELSE
		p_tyC0004Navi ACCESS ADR(tyP0800MagInfo.tyNaviLyrOff);
	END_IF

	p_tyC0005Main ACCESS ADR(tyCommon.tyMain);

	p_tyC0007Notif ACCESS ADR(tyCommon.tyNotif);

	p_tyC0008MsgBox ACCESS ADR(tyP0800MagInfo.tyMsgBoxHide);

	p_tyC0009Info ACCESS ADR(tyCommon.tyInfo);

	p_tyP0800MagInfo1 ACCESS ADR(tyP0800MagInfo.tyMagInfo1);

	p_tyP0800MagInfo2 ACCESS ADR(tyP0800MagInfo.tyMagInfo2);

	p_tyP0800MagInfo3 ACCESS ADR(tyP0800MagInfo.tyMagInfo3);

	p_tyP0800MagInfo4 ACCESS ADR(tyP0800MagInfo.tyMagInfo4);

	bDisplayMag4Info := FALSE;

END_ACTION
```

#### Act_OptP0800Navi.st
```iecst
ACTION Act_OptP0800Navi:

	IF tyP0800MagInfo.tyNaviLyr1.tyBtnBack.bRtCompl = TRUE
		OR tyP0800MagInfo.tyNaviLyr2.tyBtnBack.bRtCompl = TRUE
		THEN
		tyP0800MagInfo.tyNaviLyr1.tyBtnBack.bRtCompl	:= FALSE;
		tyP0800MagInfo.tyNaviLyr1.tyBtnBack.bValue	:= FALSE;
		tyP0800MagInfo.tyNaviLyr2.tyBtnBack.bRtCompl	:= FALSE;
		tyP0800MagInfo.tyNaviLyr2.tyBtnBack.bValue	:= FALSE;

		eChgPage	:= UIP0200OpsGen;

	ELSIF tyP0800MagInfo.tyNaviLyr1.tyBtnLeft.bRtCompl = TRUE
		OR tyP0800MagInfo.tyNaviLyr1.tyBtnRgt.bRtCompl = TRUE
		THEN
		tyP0800MagInfo.tyNaviLyr1.tyBtnLeft.bRtCompl	:= FALSE;
		tyP0800MagInfo.tyNaviLyr1.tyBtnLeft.bValue		:= FALSE;
		tyP0800MagInfo.tyNaviLyr1.tyBtnRgt.bRtCompl		:= FALSE;
		tyP0800MagInfo.tyNaviLyr1.tyBtnRgt.bValue		:= FALSE;

		p_tyC0004Navi ACCESS ADR(tyP0800MagInfo.tyNaviLyr2);

		fUIInRtStatHide(ADR(tyP0800MagInfo.tyMagInfo1.tyLyr.uiRtStat));
		fUIInRtStatHide(ADR(tyP0800MagInfo.tyMagInfo2.tyLyr.uiRtStat));
		fUIInRtStatHide(ADR(tyP0800MagInfo.tyMagInfo3.tyLyr.uiRtStat));
		fUIInRtStatOff(ADR(tyP0800MagInfo.tyMagInfo4.tyLyr.uiRtStat));

	ELSIF tyP0800MagInfo.tyNaviLyr2.tyBtnLeft.bRtCompl = TRUE
		OR tyP0800MagInfo.tyNaviLyr2.tyBtnRgt.bRtCompl = TRUE
		THEN
		tyP0800MagInfo.tyNaviLyr2.tyBtnLeft.bRtCompl	:= FALSE;
		tyP0800MagInfo.tyNaviLyr2.tyBtnLeft.bValue		:= FALSE;
		tyP0800MagInfo.tyNaviLyr2.tyBtnRgt.bRtCompl		:= FALSE;
		tyP0800MagInfo.tyNaviLyr2.tyBtnRgt.bValue		:= FALSE;

		p_tyC0004Navi ACCESS ADR(tyP0800MagInfo.tyNaviLyr1);

		fUIInRtStatOff(ADR(tyP0800MagInfo.tyMagInfo1.tyLyr.uiRtStat));
		fUIInRtStatOff(ADR(tyP0800MagInfo.tyMagInfo2.tyLyr.uiRtStat));
		fUIInRtStatOff(ADR(tyP0800MagInfo.tyMagInfo3.tyLyr.uiRtStat));
		fUIInRtStatHide(ADR(tyP0800MagInfo.tyMagInfo4.tyLyr.uiRtStat));

	END_IF

END_ACTION
```

#### Act_OptP0800Mag1Updt.st
```iecst
ACTION Act_OptP0800Mag1Updt:

	IF p_tyDI.bMagPresentSen1 THEN
		IF p_tyBuffer1BffrStat.bBffrFull THEN
			tyP0800MagInfo.tyMagInfo1.tyTxtMag1Stat.usiValueIdx	:= 2;
			tyP0800MagInfo.tyMagInfo1.tyTxtMag1Stat.usiColor	:= 0;
		ELSIF p_tyBuffer1BffrStat.bBffrMty THEN
			tyP0800MagInfo.tyMagInfo1.tyTxtMag1Stat.usiValueIdx := 1;
			tyP0800MagInfo.tyMagInfo1.tyTxtMag1Stat.usiColor	:= 1;
		ELSE
			tyP0800MagInfo.tyMagInfo1.tyTxtMag1Stat.usiValueIdx := 3;
			tyP0800MagInfo.tyMagInfo1.tyTxtMag1Stat.usiColor	:= 2;
		END_IF
	ELSE
		tyP0800MagInfo.tyMagInfo1.tyTxtMag1Stat.usiValueIdx		:= 0;
		tyP0800MagInfo.tyMagInfo1.tyTxtMag1Stat.usiColor		:= 1;
	END_IF

	//Set Magazine Empty
	IF tyP0800MagInfo.tyMagInfo1.tyBtnMag1SetEmpty.bRtCompl THEN
		tyP0800MagInfo.tyMagInfo1.tyBtnMag1SetEmpty.bValue	:= TRUE;
		IF p_bOpsMagConvLD1RlsMagAllw OR p_bOpsMagConvLD1RlsMagUmask THEN
			IF p_bPPRetSen THEN
				eBuffer1Act	:= BufferActSetMty;
			END_IF
			IF p_bOpsMagConvLD1ExtMes OR p_bOpsMagConvLD1RlsMagUmask THEN
				bEjectMag1 	:= TRUE;
				bRlsMag1 	:= TRUE;
			END_IF
		END_IF

		IF p_eBuffer1Stat = BufferActSetMty AND p_eBuffer1Status = Done THEN
			eBuffer1Act	:= BufferActIdle;
			bEjectMag1 	:= FALSE;
			bRlsMag1 	:= FALSE;
			tyP0800MagInfo.tyMagInfo1.tyBtnMag1SetEmpty.bRtCompl	:= FALSE;
			tyP0800MagInfo.tyMagInfo1.tyBtnMag1SetEmpty.bValue		:= FALSE;
		ELSIF p_bOpsRun = FALSE THEN
			tyP0800MagInfo.tyMagInfo1.tyBtnMag1SetEmpty.bRtCompl	:= FALSE;
			tyP0800MagInfo.tyMagInfo1.tyBtnMag1SetEmpty.bValue		:= FALSE;
		END_IF

	END_IF

	IF p_bOpsRun AND p_tyNtParamCurr.bProjMotorizedPullerPrep THEN
	//	tyP0800MagInfo.tyMagInfo1.tyBtnMag1SetEmpty.uiMaskRtStat.0	:= p_tyDI.bMagPresentSen1 AND (NOT p_tyBuffer1BffrStat.bBffrMty AND p_bOpsMagConvLD1RlsMagAllw)OR p_bOpsMagConvLD1RlsMagUmask;//FALSE;
		tyP0800MagInfo.tyMagInfo1.tyBtnMag1SetEmpty.uiMaskRtStat.0	:= p_tyDI.bMagPresentSen1 AND (NOT p_tyBuffer1BffrStat.bBffrMty) OR p_bOpsMagConvLD1RlsMagUmask;//FALSE;
//	ELSIF p_bOpsRun THEN
//		tyP0800MagInfo.tyMagInfo1.tyBtnMag1SetEmpty.uiMaskRtStat.0	:= FALSE;
	ELSE
		tyP0800MagInfo.tyMagInfo1.tyBtnMag1SetEmpty.uiMaskRtStat.0	:= p_tyDI.bMagPresentSen1 AND NOT p_tyBuffer1BffrStat.bBffrMty;
	END_IF

END_ACTION
```

#### Act_OptP0800Mag2Updt.st
```iecst
ACTION Act_OptP0800Mag2Updt:

	IF p_tyDI.bMagPresentSen2 THEN
		IF p_tyBuffer2BffrStat.bBffrFull THEN
			tyP0800MagInfo.tyMagInfo1.tyTxtMag2Stat.usiValueIdx	:= 2;
			tyP0800MagInfo.tyMagInfo1.tyTxtMag2Stat.usiColor	:= 0;
		ELSIF p_tyBuffer2BffrStat.bBffrMty THEN
			tyP0800MagInfo.tyMagInfo1.tyTxtMag2Stat.usiValueIdx := 1;
			tyP0800MagInfo.tyMagInfo1.tyTxtMag2Stat.usiColor	:= 1;
		ELSE
			tyP0800MagInfo.tyMagInfo1.tyTxtMag2Stat.usiValueIdx := 3;
			tyP0800MagInfo.tyMagInfo1.tyTxtMag2Stat.usiColor	:= 2;
		END_IF
	ELSE
		tyP0800MagInfo.tyMagInfo1.tyTxtMag2Stat.usiValueIdx		:= 0;
		tyP0800MagInfo.tyMagInfo1.tyTxtMag2Stat.usiColor		:= 1;
	END_IF

	//Set Magazine Empty
	IF tyP0800MagInfo.tyMagInfo1.tyBtnMag2SetEmpty.bRtCompl THEN
		tyP0800MagInfo.tyMagInfo1.tyBtnMag2SetEmpty.bValue	:= TRUE;
		IF p_bOpsMagConvLD2RlsMagAllw OR p_bOpsMagConvLD2RlsMagUmask THEN
			IF p_bPPRetSen THEN
				eBuffer2Act	:= BufferActSetMty;
			END_IF
			IF p_bOpsMagConvLD2ExtMes OR p_bOpsMagConvLD2RlsMagUmask THEN
				bEjectMag2 := TRUE;
				bRlsMag2 	:= TRUE;
			END_IF
		END_IF

		IF p_eBuffer2Stat = BufferActSetMty AND p_eBuffer2Status = Done THEN
			eBuffer2Act	:= BufferActIdle;
			bEjectMag2 := FALSE;
			bRlsMag2 	:= FALSE;
			tyP0800MagInfo.tyMagInfo1.tyBtnMag2SetEmpty.bRtCompl	:= FALSE;
			tyP0800MagInfo.tyMagInfo1.tyBtnMag2SetEmpty.bValue		:= FALSE;
		ELSIF p_bOpsRun = FALSE THEN
			tyP0800MagInfo.tyMagInfo1.tyBtnMag2SetEmpty.bRtCompl	:= FALSE;
			tyP0800MagInfo.tyMagInfo1.tyBtnMag2SetEmpty.bValue		:= FALSE;
		END_IF
	END_IF

	IF p_bOpsRun AND p_tyNtParamCurr.bProjMotorizedPullerPrep THEN
	//	tyP0800MagInfo.tyMagInfo1.tyBtnMag2SetEmpty.uiMaskRtStat.0	:= p_tyDI.bMagPresentSen2 AND (NOT p_tyBuffer2BffrStat.bBffrMty AND p_bOpsMagConvLD2RlsMagAllw) OR p_bOpsMagConvLD2RlsMagUmask;
		tyP0800MagInfo.tyMagInfo1.tyBtnMag2SetEmpty.uiMaskRtStat.0	:= p_tyDI.bMagPresentSen2 AND (NOT p_tyBuffer2BffrStat.bBffrMty) OR p_bOpsMagConvLD2RlsMagUmask;//FALSE;
//	ELSIF p_bOpsRun THEN
//		tyP0800MagInfo.tyMagInfo1.tyBtnMag2SetEmpty.uiMaskRtStat.0	:= FALSE;
	ELSE
		tyP0800MagInfo.tyMagInfo1.tyBtnMag2SetEmpty.uiMaskRtStat.0	:= p_tyDI.bMagPresentSen2 AND NOT p_tyBuffer2BffrStat.bBffrMty;
	END_IF

END_ACTION
```

#### Act_OptP0800Mag3Updt.st
```iecst
ACTION Act_OptP0800Mag3Updt:

	IF p_tyDI.bMagPresentSen3 THEN
		IF p_tyBuffer3BffrStat.bBffrFull THEN
			tyP0800MagInfo.tyMagInfo2.tyTxtMag3Stat.usiValueIdx	:= 2;
			tyP0800MagInfo.tyMagInfo2.tyTxtMag3Stat.usiColor	:= 0;
		ELSIF p_tyBuffer3BffrStat.bBffrMty THEN
			tyP0800MagInfo.tyMagInfo2.tyTxtMag3Stat.usiValueIdx := 1;
			tyP0800MagInfo.tyMagInfo2.tyTxtMag3Stat.usiColor	:= 1;
		ELSE
			tyP0800MagInfo.tyMagInfo2.tyTxtMag3Stat.usiValueIdx := 3;
			tyP0800MagInfo.tyMagInfo2.tyTxtMag3Stat.usiColor	:= 2;
		END_IF
	ELSE
		tyP0800MagInfo.tyMagInfo2.tyTxtMag3Stat.usiValueIdx		:= 0;
		tyP0800MagInfo.tyMagInfo2.tyTxtMag3Stat.usiColor		:= 1;
	END_IF

	//Set Magazine Empty
	IF tyP0800MagInfo.tyMagInfo2.tyBtnMag3SetEmpty.bRtCompl THEN
		tyP0800MagInfo.tyMagInfo2.tyBtnMag3SetEmpty.bValue	:= TRUE;
		IF p_bOpsMagConvLD3RlsMagAllw OR p_bOpsMagConvLD3RlsMagUmask THEN
			IF p_bPPRetSen THEN
				eBuffer3Act	:= BufferActSetMty;
			END_IF
			IF p_bOpsMagConvLD3ExtMes OR p_bOpsMagConvLD3RlsMagUmask THEN
				bEjectMag3 := TRUE;
				bRlsMag3 	:= TRUE;
			END_IF
		END_IF

		IF p_eBuffer3Stat = BufferActSetMty AND p_eBuffer3Status = Done THEN
			eBuffer3Act	:= BufferActIdle;
			bEjectMag3 := FALSE;
			bRlsMag3 	:= FALSE;
			tyP0800MagInfo.tyMagInfo2.tyBtnMag3SetEmpty.bRtCompl	:= FALSE;
			tyP0800MagInfo.tyMagInfo2.tyBtnMag3SetEmpty.bValue		:= FALSE;
		ELSIF p_bOpsRun = FALSE THEN
			tyP0800MagInfo.tyMagInfo2.tyBtnMag3SetEmpty.bRtCompl	:= FALSE;
			tyP0800MagInfo.tyMagInfo2.tyBtnMag3SetEmpty.bValue		:= FALSE;
		END_IF
	END_IF

	IF p_bOpsRun AND p_tyNtParamCurr.bProjMotorizedPullerPrep THEN
	//	tyP0800MagInfo.tyMagInfo2.tyBtnMag3SetEmpty.uiMaskRtStat.0	:= p_tyDI.bMagPresentSen3 AND (NOT p_tyBuffer3BffrStat.bBffrMty AND p_bOpsMagConvLD3RlsMagAllw) OR p_bOpsMagConvLD3RlsMagUmask;
		tyP0800MagInfo.tyMagInfo2.tyBtnMag3SetEmpty.uiMaskRtStat.0	:= p_tyDI.bMagPresentSen3 AND (NOT p_tyBuffer3BffrStat.bBffrMty) OR p_bOpsMagConvLD3RlsMagUmask;//FALSE;
//	ELSIF p_bOpsRun THEN
//		tyP0800MagInfo.tyMagInfo2.tyBtnMag3SetEmpty.uiMaskRtStat.0	:= FALSE;
	ELSE
		tyP0800MagInfo.tyMagInfo2.tyBtnMag3SetEmpty.uiMaskRtStat.0	:= p_tyDI.bMagPresentSen3 AND NOT p_tyBuffer3BffrStat.bBffrMty;
	END_IF

END_ACTION
```

#### Act_OptP0800Table4.st
```iecst
ACTION Act_OptP0800Table4:

	tyP0800MagInfo.tyMagInfo4.tyTable4List.tyUISlider.iMaxValue	:= DINT_TO_INT(p_tyBuffer4DispBffr.diDispIdxEnd) - (c_uiP0800TableSize - 1);

	//Call Table FB
	fbP0800Table4.sVisuNm				:= tyP0800Table4.sVisuNm;
	fbP0800Table4.udiWorkAreaStartX		:= 15;
	fbP0800Table4.udiWorkAreaEndX		:= 365;
	fbP0800Table4.udiWorkAreaStartY		:= 109;
	fbP0800Table4.udiWorkAreaEndY		:= 429;
	fbP0800Table4.udiMinXDist			:= 20;
	fbP0800Table4.udiMinYDist			:= 20;
	fbP0800Table4.uiSlideScale			:= c_uiP0800TableSize;
	fbP0800Table4.iTotalData			:= DINT_TO_INT(p_tyBuffer4DispBffr.diDispIdxEnd);
	fbP0800Table4.iTotalRow				:= c_uiP0800TableSize;
	fbP0800Table4(uiSliderStatus 		:= tyP0800MagInfo.tyMagInfo4.tyTable4List.tyUISlider.uiRtStat , a_tyUIHotspot := tyP0800MagInfo.tyMagInfo4.tyTable4List.a_tyHotspot , uiTablePos := tyP0800Table4.uiTablePos , iSliderPos := tyP0800MagInfo.tyMagInfo4.tyTable4List.tyUISlider.iValue);

	tyP0800Table4.uiSelectedRow	:= fbP0800Table4.uiSelectedRow;
	tyP0800Table4.bTableActive	:= fbP0800Table4.bTableActive;
	tyP0800Table4.bSliderActive	:= fbP0800Table4.bSliderActive;

	//Table Content
	IF p_tyDI.bMagPresentSen4 THEN
		FOR i := 1 TO c_uiP0800TableSize DO
			tyP0800MagInfo.tyMagInfo4.tyTable4List.a_tyStringDataCol0[i].sValue		:= p_tyBuffer4DispBffr.a_tyDispBffrDat[tyP0800Table4.uiTablePos + i - 1].sSltIdx;
			tyP0800MagInfo.tyMagInfo4.tyTable4List.a_tyStringDataCol1[i].sValue		:= p_tyBuffer4DispBffr.a_tyDispBffrDat[tyP0800Table4.uiTablePos + i - 1].sSltTm;
			tyP0800MagInfo.tyMagInfo4.tyTable4List.a_tyStringDataCol1[i].usiColor	:= DWORD_TO_USINT(p_tyBuffer4DispBffr.a_tyDispBffrDat[tyP0800Table4.uiTablePos + i - 1].dwColor);

		END_FOR
	ELSE
		FOR i := 1 TO c_uiP0800TableSize DO
			tyP0800MagInfo.tyMagInfo4.tyTable4List.a_tyStringDataCol0[i].sValue		:= '';
			tyP0800MagInfo.tyMagInfo4.tyTable4List.a_tyStringDataCol1[i].sValue		:= '';
			tyP0800MagInfo.tyMagInfo4.tyTable4List.a_tyStringDataCol1[i].usiColor	:= 0;

		END_FOR
	END_IF

	tyP0800MagInfo.tyMagInfo4.tyTable4List.tyUISlider.iMaxValue	:= DINT_TO_INT(p_tyBuffer4DispBffr.diDispIdxEnd) - (c_uiP0800TableSize - 1);

END_ACTION
```

#### Act_OptP0800Mag4Updt.st
```iecst
ACTION Act_OptP0800Mag4Updt:

	IF p_tyDI.bMagPresentSen4 THEN
		IF p_tyBuffer4BffrStat.bBffrFull THEN
			tyP0800MagInfo.tyMagInfo4.tyTxtMag4Stat.usiValueIdx	:= 2;
			tyP0800MagInfo.tyMagInfo4.tyTxtMag4Stat.usiColor	:= 0;
		ELSIF p_tyBuffer4BffrStat.bBffrMty THEN
			tyP0800MagInfo.tyMagInfo4.tyTxtMag4Stat.usiValueIdx := 1;
			tyP0800MagInfo.tyMagInfo4.tyTxtMag4Stat.usiColor	:= 1;
		ELSE
			tyP0800MagInfo.tyMagInfo4.tyTxtMag4Stat.usiValueIdx := 3;
			tyP0800MagInfo.tyMagInfo4.tyTxtMag4Stat.usiColor	:= 2;
		END_IF
	ELSE
		tyP0800MagInfo.tyMagInfo4.tyTxtMag4Stat.usiValueIdx		:= 0;
		tyP0800MagInfo.tyMagInfo4.tyTxtMag4Stat.usiColor		:= 1;
	END_IF

	//Set Magazine Empty
	IF tyP0800MagInfo.tyMagInfo4.tyBtnMag4SetEmpty.bRtCompl THEN
		tyP0800MagInfo.tyMagInfo4.tyBtnMag4SetEmpty.bValue	:= TRUE;

		eBuffer4Act	:= BufferActSetMty;

		IF p_eBuffer4Stat = BufferActSetMty AND p_eBuffer4Status = Done THEN
			eBuffer4Act	:= BufferActIdle;

			tyP0800MagInfo.tyMagInfo4.tyBtnMag4SetEmpty.bRtCompl	:= FALSE;
			tyP0800MagInfo.tyMagInfo4.tyBtnMag4SetEmpty.bValue		:= FALSE;
		END_IF
	END_IF

	IF p_bOpsRun THEN
		tyP0800MagInfo.tyMagInfo4.tyBtnMag4SetEmpty.uiMaskRtStat.0	:= p_tyDI.bMagPresentSen4 AND NOT p_tyBuffer4BffrStat.bBffrMty AND p_bOpsMagConvLD4RlsMagAllw;
	ELSE
		tyP0800MagInfo.tyMagInfo4.tyBtnMag4SetEmpty.uiMaskRtStat.0	:= p_tyDI.bMagPresentSen4 AND NOT p_tyBuffer4BffrStat.bBffrMty;
	END_IF

END_ACTION
```

#### Act_EntP0900Disp.st
```iecst
ACTION Act_EntP0900Disp:

	//Access Address
	p_tyC0005Main ACCESS ADR(tyCommon.tyMain);

	p_tyC0007Notif ACCESS ADR(tyCommon.tyNotif);

	p_tyC0008MsgBox ACCESS ADR(tyP0900GenIn.tyMsgBoxHide);

	p_tyC0009Info ACCESS ADR(tyCommon.tyInfo);

	p_tyP0900GenIn1 ACCESS ADR(tyP0900GenIn.tyGenIn1);
	p_tyP0900GenIn2 ACCESS ADR(tyP0900GenIn.tyGenIn2);

END_ACTION
```

#### Act_OptP0900ReadDI.st
```iecst
ACTION Act_OptP0900ReadDI:

	tyP0900GenIn.tyGenIn1.tyBtnSafetyRly.bValue				:= p_tyDI.bSafetyRlySig;
	tyP0900GenIn.tyGenIn1.tyBtnEStop.bValue					:= p_tyDI.bEStopSig;
	tyP0900GenIn.tyGenIn1.tyBtnCoverSW.bValue				:= p_tyDI.bCoverSWSig;
	tyP0900GenIn.tyGenIn1.tyBtnLifterTimingBeltSen.bValue	:= p_tyDI.bLifterTimingBeltSen;
	tyP0900GenIn.tyGenIn1.tyBtnLifterSafetyLmtSW1.bValue	:= p_tyDI.bLifterSafetyLmtSW1;
	tyP0900GenIn.tyGenIn1.tyBtnLifterSafetyLmtSW2.bValue	:= p_tyDI.bLifterSafetyLmtSW2;
	tyP0900GenIn.tyGenIn1.tyBtnMag1PresentSen.bValue		:= p_tyDI.bMagPresentSen1;
	tyP0900GenIn.tyGenIn1.tyBtnMag2PresentSen.bValue		:= p_tyDI.bMagPresentSen2;
	tyP0900GenIn.tyGenIn1.tyBtnMag3PresentSen.bValue		:= p_tyDI.bMagPresentSen3;
	tyP0900GenIn.tyGenIn1.tyBtnMag4PresentSen.bValue		:= p_tyDI.bMagPresentSen4;
	tyP0900GenIn.tyGenIn1.tyBtnCurtainSafetyRly.bValue		:= p_tyDI.bCurtainSafetySig2;
	tyP0900GenIn.tyGenIn1.tyBtnMagWidthChk.bValue		:= p_tyDI.bMagWidthChkSen;

	tyP0900GenIn.tyGenIn2.tyBtnMag1OrientationChkSen1.bValue	:= p_tyDI.bMag1OrientChkSen1;
	tyP0900GenIn.tyGenIn2.tyBtnMag1OrientationChkSen2.bValue	:= p_tyDI.bMag1OrientChkSen2;
	tyP0900GenIn.tyGenIn2.tyBtnMag2OrientationChkSen1.bValue	:= p_tyDI.bMag2OrientChkSen1;
	tyP0900GenIn.tyGenIn2.tyBtnMag2OrientationChkSen2.bValue	:= p_tyDI.bMag2OrientChkSen2;
	tyP0900GenIn.tyGenIn2.tyBtnMag3OrientationChkSen1.bValue	:= p_tyDI.bMag3OrientChkSen1;
	tyP0900GenIn.tyGenIn2.tyBtnMag3OrientationChkSen2.bValue	:= p_tyDI.bMag3OrientChkSen2;
	tyP0900GenIn.tyGenIn2.tyBtnMag4OrientationChkSen1.bValue	:= p_tyDI.bMag4OrientChkSen1;
	tyP0900GenIn.tyGenIn2.tyBtnMag4OrientationChkSen2.bValue	:= p_tyDI.bMag4OrientChkSen2;
END_ACTION
```

#### Act_EntP0910Disp.st
```iecst
ACTION Act_EntP0910Disp:

	//Access Address
	p_tyC0005Main ACCESS ADR(tyCommon.tyMain);

	p_tyC0007Notif ACCESS ADR(tyCommon.tyNotif);

	p_tyC0008MsgBox ACCESS ADR(tyP0910GenOut.tyMsgBoxHide);

	p_tyC0009Info ACCESS ADR(tyCommon.tyInfo);

	p_tyP0910GenOut ACCESS ADR(tyP0910GenOut.tyGenOut);

	p_tyP0910GenOutCurtainSen ACCESS ADR(tyP0910GenOut.tyGenOutCurtainSen);

END_ACTION
```

#### Act_OptP0910RstMnl.st
```iecst
ACTION Act_OptP0910RstMnl:

	IF EDGEPOS((bUIManualMod = FALSE) OR (p_eRstErrStatus = Error)) THEN
		eRstErrAct	:= RstErrActIdle;

		tyP0910GenOut.tyGenOut.tyBtnSafetyRst.bValue	:= FALSE;

		//curtain sensor
		tyP0910GenOut.tyGenOutCurtainSen.tyBtnRstCurtainSen.bRtCompl	:= FALSE;
		tyP0910GenOut.tyGenOutCurtainSen.tyBtnRstCurtainSen.bValue   	:= FALSE;
		//	bSafetyCurtainReset	:= FALSE;
		tyP0910GenOut.tyGenOutCurtainSen.tyBtnBypCurtainSenPBLED.bValue	:= FALSE;
		bBypCurtainPBLED	:= FALSE;

		tyP0910GenOut.tyGenOutCurtainSen.tyBtnBypCurtainSen.bValue	:= FALSE;
		bBypCurtainSen	:= FALSE;
		//bSafetyCurtainReset := FALSE;

	END_IF

	IF EDGEPOS((bUIManualMod = FALSE) OR (p_eTLBuzStatus = Error)) THEN
		eTLBuzAct	:= TLBuzActIdle;

		tyP0910GenOut.tyGenOut.tyBtnTLGreen.bValue		:= FALSE;
		tyP0910GenOut.tyGenOut.tyBtnTLAmber.bValue		:= FALSE;
		tyP0910GenOut.tyGenOut.tyBtnTLRed.bValue		:= FALSE;
		tyP0910GenOut.tyGenOut.tyBtnBuzzer.bValue		:= FALSE;
	END_IF

END_ACTION
```

#### Act_OptP0910WriteDO.st
```iecst
ACTION Act_OptP0910WriteDO:

	//TL Safety Relay
	IF tyP0910GenOut.tyGenOut.tyBtnSafetyRst.bRtCompl = TRUE THEN
		IF tyP0910GenOut.tyGenOut.tyBtnSafetyRst.bValue = TRUE THEN
			eRstErrAct	:= RstErrActSetSafetyRlyRst;

			IF p_eRstErrStat = RstErrActSetSafetyRlyRst AND p_eRstErrStatus = Done THEN
				eRstErrAct	:= RstErrActIdle;

				tyP0910GenOut.tyGenOut.tyBtnSafetyRst.bRtCompl	:= FALSE;
			END_IF
		ELSE
			eRstErrAct	:= RstErrActRstSafetyRlyRst;

			IF p_eRstErrStat = RstErrActRstSafetyRlyRst AND p_eRstErrStatus = Done THEN
				eRstErrAct	:= RstErrActIdle;

				tyP0910GenOut.tyGenOut.tyBtnSafetyRst.bRtCompl	:= FALSE;
			END_IF

		END_IF
	END_IF

	// TL Green
	IF tyP0910GenOut.tyGenOut.tyBtnTLGreen.bRtCompl = TRUE THEN
		IF tyP0910GenOut.tyGenOut.tyBtnTLGreen.bValue = TRUE THEN
			eTLBuzAct	:= TLBuzActSetGreen;

			IF p_eTLBuzStat = TLBuzActSetGreen AND p_eTLBuzStatus = Done THEN
				eTLBuzAct	:= TLBuzActIdle;

				tyP0910GenOut.tyGenOut.tyBtnTLGreen.bRtCompl	:= FALSE;
			END_IF
		ELSE
			eTLBuzAct	:= TLBuzActRstGreen;

			IF p_eTLBuzStat = TLBuzActRstGreen AND p_eTLBuzStatus = Done THEN
				eTLBuzAct	:= TLBuzActIdle;

				tyP0910GenOut.tyGenOut.tyBtnTLGreen.bRtCompl	:= FALSE;
			END_IF

		END_IF
	END_IF

	//TL Amber
	IF tyP0910GenOut.tyGenOut.tyBtnTLAmber.usiTxtIdx = 0 THEN
		IF tyP0910GenOut.tyGenOut.tyBtnTLAmber.bRtCompl = TRUE THEN
			IF tyP0910GenOut.tyGenOut.tyBtnTLAmber.bValue = TRUE THEN
				eTLBuzAct	:= TLBuzActSetAmber;

				IF p_eTLBuzStat = TLBuzActSetAmber AND p_eTLBuzStatus = Done THEN
					eTLBuzAct	:= TLBuzActIdle;

					tyP0910GenOut.tyGenOut.tyBtnTLAmber.bRtCompl	:= FALSE;
				END_IF
			ELSE
				eTLBuzAct	:= TLBuzActRstAmber;

				IF p_eTLBuzStat = TLBuzActRstAmber AND p_eTLBuzStatus = Done THEN
					eTLBuzAct	:= TLBuzActIdle;

					tyP0910GenOut.tyGenOut.tyBtnTLAmber.bRtCompl	:= FALSE;
				END_IF

			END_IF
		END_IF
	ELSIF tyP0910GenOut.tyGenOut.tyBtnTLAmber.usiTxtIdx = 2 THEN // white
		IF tyP0910GenOut.tyGenOut.tyBtnTLAmber.bRtCompl = TRUE THEN
			IF tyP0910GenOut.tyGenOut.tyBtnTLAmber.bValue = TRUE THEN
				eTLBuzAct	:= TLBuzActSetWhite;

				IF p_eTLBuzStat = TLBuzActSetWhite AND p_eTLBuzStatus = Done THEN
					eTLBuzAct	:= TLBuzActIdle;

					tyP0910GenOut.tyGenOut.tyBtnTLAmber.bRtCompl	:= FALSE;
				END_IF
			ELSE
				eTLBuzAct	:= TLBuzActRstWhite;

				IF p_eTLBuzStat = TLBuzActRstWhite AND p_eTLBuzStatus = Done THEN
					eTLBuzAct	:= TLBuzActIdle;

					tyP0910GenOut.tyGenOut.tyBtnTLAmber.bRtCompl	:= FALSE;
				END_IF

			END_IF
		END_IF
	END_IF
	//TL Red
	IF tyP0910GenOut.tyGenOut.tyBtnTLRed.bRtCompl = TRUE THEN
		IF tyP0910GenOut.tyGenOut.tyBtnTLRed.bValue = TRUE THEN
			eTLBuzAct	:= TLBuzActSetRed;

			IF p_eTLBuzStat = TLBuzActSetRed AND p_eTLBuzStatus = Done THEN
				eTLBuzAct	:= TLBuzActIdle;

				tyP0910GenOut.tyGenOut.tyBtnTLRed.bRtCompl	:= FALSE;
			END_IF
		ELSE
			eTLBuzAct	:= TLBuzActRstRed;

			IF p_eTLBuzStat = TLBuzActRstRed AND p_eTLBuzStatus = Done THEN
				eTLBuzAct	:= TLBuzActIdle;

				tyP0910GenOut.tyGenOut.tyBtnTLRed.bRtCompl	:= FALSE;
			END_IF

		END_IF
	END_IF

	//TL Buzzer
	IF tyP0910GenOut.tyGenOut.tyBtnBuzzer.bRtCompl = TRUE THEN
		IF tyP0910GenOut.tyGenOut.tyBtnBuzzer.bValue = TRUE THEN
			eTLBuzAct	:= TLBuzActSetBuz;

			IF p_eTLBuzStat = TLBuzActSetBuz AND p_eTLBuzStatus = Done THEN
				eTLBuzAct	:= TLBuzActIdle;

				tyP0910GenOut.tyGenOut.tyBtnBuzzer.bRtCompl	:= FALSE;
			END_IF
		ELSE
			eTLBuzAct	:= TLBuzActRstBuz;

			IF p_eTLBuzStat = TLBuzActRstBuz AND p_eTLBuzStatus = Done THEN
				eTLBuzAct	:= TLBuzActIdle;

				tyP0910GenOut.tyGenOut.tyBtnBuzzer.bRtCompl	:= FALSE;
			END_IF

		END_IF
	END_IF

//	IF tyP0910GenOut.tyGenOut.tyBtnSafetyCurtainRst.bRtCompl = TRUE THEN
//
//		IF tyP0910GenOut.tyGenOut.tyBtnSafetyCurtainRst.bValue = TRUE THEN
//			bSafetyCurtainReset := TRUE;
//			tyP0910GenOut.tyGenOut.tyBtnSafetyCurtainRst.bRtCompl := FALSE;
//		ELSE
//			bSafetyCurtainReset := FALSE;
//			tyP0910GenOut.tyGenOut.tyBtnSafetyCurtainRst.bRtCompl := FALSE;
//		END_IF
//	END_IF

	IF tyP0910GenOut.tyGenOutCurtainSen.tyBtnRstCurtainSen.bRtCompl = TRUE THEN

		IF tyP0910GenOut.tyGenOutCurtainSen.tyBtnRstCurtainSen.bValue = TRUE THEN
			bSafetyCurtainReset := TRUE;
			tyP0910GenOut.tyGenOutCurtainSen.tyBtnRstCurtainSen.bRtCompl := FALSE;
		ELSE
			bSafetyCurtainReset := FALSE;
			tyP0910GenOut.tyGenOutCurtainSen.tyBtnRstCurtainSen.bRtCompl := FALSE;
		END_IF
	END_IF

	bBypCurtainPBLED	:= tyP0910GenOut.tyGenOutCurtainSen.tyBtnBypCurtainSenPBLED.bValue;
	bBypCurtainSen		:= tyP0910GenOut.tyGenOutCurtainSen.tyBtnBypCurtainSen.bValue;

END_ACTION
```

#### Act_EntP0920Disp.st
```iecst
ACTION Act_EntP0920Disp:

	//Access Address
	p_tyC0002FullMask ACCESS ADR(tyP0920MtrNPneuCtrl.tyFullMaskHide);

	p_tyC0005Main ACCESS ADR(tyCommon.tyMain);

	p_tyC0007Notif ACCESS ADR(tyCommon.tyNotif);

	p_tyC0008MsgBox ACCESS ADR(tyP0920MtrNPneuCtrl.tyMsgBoxHide);

	p_tyC0009Info ACCESS ADR(tyCommon.tyInfo);

	p_tyP0920MtrNPneuCtrl ACCESS ADR(tyP0920MtrNPneuCtrl.tyMtrNPneuCtrl);
	p_tyP0920MtrNPneuCtrlPneu ACCESS ADR(tyP0920MtrNPneuCtrl.tyMtrNPneuCtrlPneu);

	//Display
	//Auto Width
	tyP0920MtrNPneuCtrl.tyMtrNPneuCtrl.tyBtnAW.uiMaskRtStat.0		:= NOT(p_tyNtParamCurr.bAWPrep AND p_tyMcParamCurr.bAWDis);
	tyP0920MtrNPneuCtrl.tyMtrNPneuCtrl.tyBtnAWPushPul.uiMaskRtStat.0:= NOT(p_tyNtParamCurr.bAWPrep AND p_tyMcParamCurr.bAWPusherDis);

END_ACTION
```

#### Act_OptP0920ChgPage.st
```iecst
ACTION Act_OptP0920ChgPage:

	IF tyP0920MtrNPneuCtrl.tyMtrNPneuCtrlPneu.tyBtnShutter.bRtCompl THEN
		tyP0920MtrNPneuCtrl.tyMtrNPneuCtrlPneu.tyBtnShutter.bRtCompl	:= FALSE;
		tyP0920MtrNPneuCtrl.tyMtrNPneuCtrlPneu.tyBtnShutter.bValue		:= FALSE;
		eChgPage														:= UIP0921Shutter;

	ELSIF tyP0920MtrNPneuCtrl.tyMtrNPneuCtrl.tyBtnMag1Conv.bRtCompl AND bDispMagConv1 THEN
		tyP0920MtrNPneuCtrl.tyMtrNPneuCtrl.tyBtnMag1Conv.bRtCompl		:= FALSE;
		tyP0920MtrNPneuCtrl.tyMtrNPneuCtrl.tyBtnMag1Conv.bValue			:= FALSE;
		eChgPage														:= UIP0930MagConv1;

	ELSIF tyP0920MtrNPneuCtrl.tyMtrNPneuCtrl.tyBtnMag1Conv.bRtCompl AND bDispMagConv2 THEN
		tyP0920MtrNPneuCtrl.tyMtrNPneuCtrl.tyBtnMag1Conv.bRtCompl		:= FALSE;
		tyP0920MtrNPneuCtrl.tyMtrNPneuCtrl.tyBtnMag1Conv.bValue			:= FALSE;
		eChgPage														:= UIP0931MagConv2;

	ELSIF tyP0920MtrNPneuCtrl.tyMtrNPneuCtrl.tyBtnMag1Conv.bRtCompl AND bDispMagConv3 THEN
		tyP0920MtrNPneuCtrl.tyMtrNPneuCtrl.tyBtnMag1Conv.bRtCompl		:= FALSE;
		tyP0920MtrNPneuCtrl.tyMtrNPneuCtrl.tyBtnMag1Conv.bValue			:= FALSE;
		eChgPage														:= UIP0932MagConv3;

	ELSIF tyP0920MtrNPneuCtrl.tyMtrNPneuCtrl.tyBtnMag1Conv.bRtCompl AND bDispMagConv4 THEN
		tyP0920MtrNPneuCtrl.tyMtrNPneuCtrl.tyBtnMag1Conv.bRtCompl		:= FALSE;
		tyP0920MtrNPneuCtrl.tyMtrNPneuCtrl.tyBtnMag1Conv.bValue			:= FALSE;
		eChgPage														:= UIP0939MagConv4;

	ELSIF tyP0920MtrNPneuCtrl.tyMtrNPneuCtrl.tyBtnPullerConv.bRtCompl = TRUE THEN
		tyP0920MtrNPneuCtrl.tyMtrNPneuCtrl.tyBtnPullerConv.bRtCompl		:= FALSE;
		tyP0920MtrNPneuCtrl.tyMtrNPneuCtrl.tyBtnPullerConv.bValue		:= FALSE;
		eChgPage														:= UIP0933PullConv;

	ELSIF tyP0920MtrNPneuCtrl.tyMtrNPneuCtrl.tyBtnAW.bRtCompl = TRUE THEN
		tyP0920MtrNPneuCtrl.tyMtrNPneuCtrl.tyBtnAW.bRtCompl				:= FALSE;
		tyP0920MtrNPneuCtrl.tyMtrNPneuCtrl.tyBtnAW.bValue				:= FALSE;
		eChgPage														:= UIP0934AW;

	ELSIF tyP0920MtrNPneuCtrl.tyMtrNPneuCtrl.tyBtnLifter.bRtCompl = TRUE THEN
		tyP0920MtrNPneuCtrl.tyMtrNPneuCtrl.tyBtnLifter.bRtCompl			:= FALSE;
		tyP0920MtrNPneuCtrl.tyMtrNPneuCtrl.tyBtnLifter.bValue			:= FALSE;
		eChgPage														:= UIP0935Lifter;

	ELSIF tyP0920MtrNPneuCtrl.tyMtrNPneuCtrl.tyBtnTrav.bRtCompl = TRUE THEN
		tyP0920MtrNPneuCtrl.tyMtrNPneuCtrl.tyBtnTrav.bRtCompl			:= FALSE;
		tyP0920MtrNPneuCtrl.tyMtrNPneuCtrl.tyBtnTrav.bValue				:= FALSE;
		eChgPage														:= UIP0936Trav;

	ELSIF tyP0920MtrNPneuCtrl.tyMtrNPneuCtrl.tyBtnAWPushPul.bRtCompl = TRUE THEN
		tyP0920MtrNPneuCtrl.tyMtrNPneuCtrl.tyBtnAWPushPul.bRtCompl		:= FALSE;
		tyP0920MtrNPneuCtrl.tyMtrNPneuCtrl.tyBtnAWPushPul.bValue		:= FALSE;
		eChgPage														:= UIP0937AWPushOrPuller;

	ELSIF tyP0920MtrNPneuCtrl.tyMtrNPneuCtrlPneu.tyBtnSafetyBar.bRtCompl THEN
		tyP0920MtrNPneuCtrl.tyMtrNPneuCtrlPneu.tyBtnSafetyBar.bRtCompl	:= FALSE;
		tyP0920MtrNPneuCtrl.tyMtrNPneuCtrlPneu.tyBtnSafetyBar.bValue	:= FALSE;
		eChgPage														:= UIP0923SafetyBar;

	ELSIF tyP0920MtrNPneuCtrl.tyMtrNPneuCtrlPneu.tyBtnTrolleyLck.bRtCompl THEN
		tyP0920MtrNPneuCtrl.tyMtrNPneuCtrlPneu.tyBtnTrolleyLck.bRtCompl	:= FALSE;
		tyP0920MtrNPneuCtrl.tyMtrNPneuCtrlPneu.tyBtnTrolleyLck.bValue	:= FALSE;
		eChgPage														:= UIP0924TrolleyLck;
	END_IF

END_ACTION
```

#### Act_EntP0921Disp.st
```iecst
ACTION Act_EntP0921Disp:

	//Access Address
	p_tyC0003DualMask ACCESS ADR(tyP0921InletNOutletShutter.tyDualMaskHide);

	IF p_tyNtParamCurr.tyDISettings.diInShutterOpenRS2 > 0 AND p_tyNtParamCurr.tyDISettings.diInShutterOpenRS3 > 0 THEN
		p_tyC0004Navi ACCESS ADR(tyP0921InletNOutletShutter.tyNaviLyr1);
	ELSIF p_tyNtParamCurr.bProjOutShutter2Prep THEN
		p_tyC0004Navi ACCESS ADR(tyP0921InletNOutletShutter.tyNaviOutlet21);
		tyP0921InletNOutletShutter.tyInletShutterCom.tyLyr.uiRtStat := FALSE;
		tyP0921InletNOutletShutter.tyInletShutterFB.tyLyr.uiRtStat := FALSE;
	ELSE
		p_tyC0004Navi ACCESS ADR(tyP0921InletNOutletShutter.tyNaviBack);
	END_IF

	p_tyC0005Main ACCESS ADR(tyCommon.tyMain);

	p_tyC0007Notif ACCESS ADR(tyCommon.tyNotif);

	p_tyC0008MsgBox ACCESS ADR(tyP0921InletNOutletShutter.tyMsgBoxHide);

	p_tyC0009Info ACCESS ADR(tyCommon.tyInfo);

	p_tyP0921InletShutterCom ACCESS ADR(tyP0921InletNOutletShutter.tyInletShutterCom);
	p_tyP0921InletShutterDC ACCESS ADR(tyP0921InletNOutletShutter.tyInletShutterDC);
	p_tyP0921InletShutterFB ACCESS ADR(tyP0921InletNOutletShutter.tyInletShutterFB);

	p_tyP0921OutletShutterCom ACCESS ADR(tyP0921InletNOutletShutter.tyOutletShutterCom);
	p_tyP0921OutletShutterDC ACCESS ADR(tyP0921InletNOutletShutter.tyOutletShutterDC);
	p_tyP0921OutletShutterFB ACCESS ADR(tyP0921InletNOutletShutter.tyOutletShutterFB);
	p_tyP0921OutletShutterDis ACCESS ADR(tyP0921InletNOutletShutter.tyOutletShutterDis);

	//Display
	tyP0921InletNOutletShutter.tyOutletShutterDis.tyLyr.uiRtStat.0	:= TRUE;//NOT(p_tyNtParamCurr.bProjOutletShutPrep AND p_tyMcParamCurr.bOutShutterDis);

	//Display
//	tyP0921InletNOutletShutter.tyInletShutterCom.tyLyr.uiRtStat.0	:= NOT(p_tyNtParamCurr.bProjInletShutPrep);
//	tyP0921InletNOutletShutter.tyInletShutterDC.tyLyr.uiRtStat.0	:= TRUE;
//	tyP0921InletNOutletShutter.tyInletShutterFB.tyLyr.uiRtStat.0	:= NOT(p_tyNtParamCurr.bProjInletShutPrep);
//
//	tyP0921InletNOutletShutter.tyOutletShutterCom.tyLyr.uiRtStat.0	:= NOT(p_tyNtParamCurr.bProjOutletShutPrep);
//	tyP0921InletNOutletShutter.tyOutletShutterDC.tyLyr.uiRtStat.0	:= TRUE;
//	tyP0921InletNOutletShutter.tyOutletShutterFB.tyLyr.uiRtStat.0	:= NOT(p_tyNtParamCurr.bProjOutletShutPrep);

END_ACTION
```

#### Act_OptP0921Navi.st
```iecst
ACTION Act_OptP0921Navi:

	IF tyP0921InletNOutletShutter.tyNaviBack.tyBtnBack.bRtCompl = TRUE THEN
		eChgPage		:= UIP0920MtrNPneuCtrl;

		tyP0921InletNOutletShutter.tyNaviBack.tyBtnBack.bRtCompl 	:= FALSE;
		tyP0921InletNOutletShutter.tyNaviBack.tyBtnBack.bValue		:= FALSE;

	ELSIF tyP0921InletNOutletShutter.tyNaviLyr1.tyBtnBack.bRtCompl = TRUE OR tyP0921InletNOutletShutter.tyNaviLyr2.tyBtnBack.bRtCompl = TRUE OR
		tyP0921InletNOutletShutter.tyNaviOutlet21.tyBtnBack.bRtCompl OR	tyP0921InletNOutletShutter.tyNaviOutlet22.tyBtnBack.bRtCompl THEN

		eChgPage		:= UIP0920MtrNPneuCtrl;

		tyP0921InletNOutletShutter.tyNaviLyr1.tyBtnBack.bRtCompl := FALSE;
		tyP0921InletNOutletShutter.tyNaviLyr1.tyBtnBack.bValue	 := FALSE;
		tyP0921InletNOutletShutter.tyNaviLyr2.tyBtnBack.bRtCompl := FALSE;
		tyP0921InletNOutletShutter.tyNaviLyr2.tyBtnBack.bValue	 := FALSE;

		tyP0921InletNOutletShutter.tyNaviOutlet21.tyBtnBack.bRtCompl := FALSE;
		tyP0921InletNOutletShutter.tyNaviOutlet21.tyBtnBack.bValue	 := FALSE;
		tyP0921InletNOutletShutter.tyNaviOutlet22.tyBtnBack.bRtCompl := FALSE;
		tyP0921InletNOutletShutter.tyNaviOutlet22.tyBtnBack.bValue	 := FALSE;

	ELSIF tyP0921InletNOutletShutter.tyNaviLyr1.tyBtnRgt.bRtCompl THEN

		p_tyC0004Navi ACCESS ADR (tyP0921InletNOutletShutter.tyNaviLyr2);

		p_tyP0921InletShutterCom ACCESS ADR(tyP0921InletNOutletShutter.tyInletShutterCom2);
		p_tyP0921InletShutterDC ACCESS ADR(tyP0921InletNOutletShutter.tyInletShutterDC2);
		p_tyP0921InletShutterFB ACCESS ADR(tyP0921InletNOutletShutter.tyInletShutterFB2);
//		p_tyP0921InletShutterDis ACCESS ADR(tyP0921InletNOutletShutter.tyInletShutterDis2);

		p_tyP0921OutletShutterCom ACCESS ADR(tyP0921InletNOutletShutter.tyInletShutterCom3);
		p_tyP0921OutletShutterDC ACCESS ADR(tyP0921InletNOutletShutter.tyInletShutterDC3);
		p_tyP0921OutletShutterFB ACCESS ADR(tyP0921InletNOutletShutter.tyInletShutterFB3);
		p_tyP0921OutletShutterDis ACCESS ADR(tyP0921InletNOutletShutter.tyOutletShutterDis);

		tyP0921InletNOutletShutter.tyInletShutterDC2.tyBtnOpen2.uiRtStat := TRUE;
		tyP0921InletNOutletShutter.tyInletShutterDC2.tyBtnOpen3.uiRtStat := TRUE;
		tyP0921InletNOutletShutter.tyOutletShutterDis.tyLyr.uiRtStat.0 := TRUE;
		tyP0921InletNOutletShutter.tyNaviLyr1.tyBtnRgt.bRtCompl := FALSE;
		tyP0921InletNOutletShutter.tyNaviLyr1.tyBitmapPageDisp.usiValueIdx :=2;
		tyP0921InletNOutletShutter.tyNaviLyr2.tyBitmapPageDisp.usiValueIdx :=2;

	ELSIF tyP0921InletNOutletShutter.tyNaviLyr1.tyBtnLeft.bRtCompl THEN

		p_tyC0004Navi ACCESS ADR (tyP0921InletNOutletShutter.tyNaviLyr2);

		p_tyP0921InletShutterCom ACCESS ADR(tyP0921InletNOutletShutter.tyInletShutterCom2);
		p_tyP0921InletShutterDC ACCESS ADR(tyP0921InletNOutletShutter.tyInletShutterDC2);
		p_tyP0921InletShutterFB ACCESS ADR(tyP0921InletNOutletShutter.tyInletShutterFB2);
	//	p_tyP0921InletShutterDis ACCESS ADR(tyP0921InletNOutletShutter.tyInletShutterDis2);

		p_tyP0921OutletShutterCom ACCESS ADR(tyP0921InletNOutletShutter.tyInletShutterCom3);
		p_tyP0921OutletShutterDC ACCESS ADR(tyP0921InletNOutletShutter.tyInletShutterDC3);
		p_tyP0921OutletShutterFB ACCESS ADR(tyP0921InletNOutletShutter.tyInletShutterFB3);
		p_tyP0921OutletShutterDis ACCESS ADR(tyP0921InletNOutletShutter.tyOutletShutterDis);

		tyP0921InletNOutletShutter.tyInletShutterDC2.tyBtnOpen2.uiRtStat := TRUE;
		tyP0921InletNOutletShutter.tyInletShutterDC2.tyBtnOpen3.uiRtStat := TRUE;
		tyP0921InletNOutletShutter.tyOutletShutterDis.tyLyr.uiRtStat.0 := TRUE;
		tyP0921InletNOutletShutter.tyNaviLyr1.tyBtnLeft.bRtCompl := FALSE;
		tyP0921InletNOutletShutter.tyNaviLyr1.tyBitmapPageDisp.usiValueIdx :=2;
		tyP0921InletNOutletShutter.tyNaviLyr2.tyBitmapPageDisp.usiValueIdx :=2;

	ELSIF tyP0921InletNOutletShutter.tyNaviLyr2.tyBtnRgt.bRtCompl OR tyP0921InletNOutletShutter.tyNaviOutlet22.tyBtnRgt.bRtCompl THEN
		IF tyP0921InletNOutletShutter.tyNaviLyr2.tyBtnRgt.bRtCompl THEN
			p_tyC0004Navi ACCESS ADR (tyP0921InletNOutletShutter.tyNaviLyr1);
		ELSIF tyP0921InletNOutletShutter.tyNaviOutlet22.tyBtnRgt.bRtCompl THEN
			p_tyC0004Navi ACCESS ADR (tyP0921InletNOutletShutter.tyNaviOutlet21);
			tyP0921InletNOutletShutter.tyOutletShutterCom.tyTxtTit.usiValueIdx := 148-6; //6
			tyP0921InletNOutletShutter.tyInletShutterCom.tyLyr.uiRtStat := FALSE;
			tyP0921InletNOutletShutter.tyInletShutterFB.tyLyr.uiRtStat := FALSE;
		END_IF

		p_tyP0921InletShutterCom ACCESS ADR(tyP0921InletNOutletShutter.tyInletShutterCom);
		p_tyP0921InletShutterDC ACCESS ADR(tyP0921InletNOutletShutter.tyInletShutterDC);
		p_tyP0921InletShutterFB ACCESS ADR(tyP0921InletNOutletShutter.tyInletShutterFB);

		p_tyP0921OutletShutterCom ACCESS ADR(tyP0921InletNOutletShutter.tyOutletShutterCom);
		p_tyP0921OutletShutterDC ACCESS ADR(tyP0921InletNOutletShutter.tyOutletShutterDC);
		p_tyP0921OutletShutterFB ACCESS ADR(tyP0921InletNOutletShutter.tyOutletShutterFB);
		p_tyP0921OutletShutterDis ACCESS ADR(tyP0921InletNOutletShutter.tyOutletShutterDis);

		tyP0921InletNOutletShutter.tyOutletShutterDis.tyLyr.uiRtStat.0	:= TRUE;//NOT(p_tyNtParamCurr.bProjOutletShutPrep AND p_tyMcParamCurr.bOutShutterDis);
		tyP0921InletNOutletShutter.tyNaviLyr2.tyBtnRgt.bRtCompl := FALSE;
		tyP0921InletNOutletShutter.tyNaviLyr1.tyBitmapPageDisp.usiValueIdx :=1;
		tyP0921InletNOutletShutter.tyNaviLyr2.tyBitmapPageDisp.usiValueIdx :=1;

		tyP0921InletNOutletShutter.tyNaviOutlet22.tyBtnRgt.bRtCompl := FALSE;
		tyP0921InletNOutletShutter.tyNaviOutlet21.tyBitmapPageDisp.usiValueIdx :=1;
		tyP0921InletNOutletShutter.tyNaviOutlet22.tyBitmapPageDisp.usiValueIdx :=1;

	ELSIF tyP0921InletNOutletShutter.tyNaviLyr2.tyBtnLeft.bRtCompl OR tyP0921InletNOutletShutter.tyNaviOutlet22.tyBtnLeft.bRtCompl THEN
		IF tyP0921InletNOutletShutter.tyNaviLyr2.tyBtnLeft.bRtCompl THEN
			p_tyC0004Navi ACCESS ADR (tyP0921InletNOutletShutter.tyNaviLyr1);
		ELSIF tyP0921InletNOutletShutter.tyNaviOutlet22.tyBtnLeft.bRtCompl THEN
			p_tyC0004Navi ACCESS ADR (tyP0921InletNOutletShutter.tyNaviOutlet21);
			tyP0921InletNOutletShutter.tyOutletShutterCom.tyTxtTit.usiValueIdx := 148-6; //6
			tyP0921InletNOutletShutter.tyInletShutterCom.tyLyr.uiRtStat := FALSE;
			tyP0921InletNOutletShutter.tyInletShutterFB.tyLyr.uiRtStat := FALSE;
		END_IF

		p_tyP0921InletShutterCom ACCESS ADR(tyP0921InletNOutletShutter.tyInletShutterCom);
		p_tyP0921InletShutterDC ACCESS ADR(tyP0921InletNOutletShutter.tyInletShutterDC);
		p_tyP0921InletShutterFB ACCESS ADR(tyP0921InletNOutletShutter.tyInletShutterFB);
	//	p_tyP0921InletShutterDis ACCESS ADR(tyP0921InletNOutletShutter.tyInletShutterDis);

		p_tyP0921OutletShutterCom ACCESS ADR(tyP0921InletNOutletShutter.tyOutletShutterCom);
		p_tyP0921OutletShutterDC ACCESS ADR(tyP0921InletNOutletShutter.tyOutletShutterDC);
		p_tyP0921OutletShutterFB ACCESS ADR(tyP0921InletNOutletShutter.tyOutletShutterFB);
		p_tyP0921OutletShutterDis ACCESS ADR(tyP0921InletNOutletShutter.tyOutletShutterDis);

		tyP0921InletNOutletShutter.tyOutletShutterDis.tyLyr.uiRtStat.0	:= TRUE;//NOT(p_tyNtParamCurr.bProjOutletShutPrep AND p_tyMcParamCurr.bOutShutterDis);
		tyP0921InletNOutletShutter.tyNaviLyr2.tyBtnLeft.bRtCompl := FALSE;
		tyP0921InletNOutletShutter.tyNaviLyr1.tyBitmapPageDisp.usiValueIdx :=1;
		tyP0921InletNOutletShutter.tyNaviLyr2.tyBitmapPageDisp.usiValueIdx :=1;

		tyP0921InletNOutletShutter.tyNaviOutlet22.tyBtnLeft.bRtCompl := FALSE;
		tyP0921InletNOutletShutter.tyNaviOutlet21.tyBitmapPageDisp.usiValueIdx :=1;
		tyP0921InletNOutletShutter.tyNaviOutlet22.tyBitmapPageDisp.usiValueIdx :=1;

	ELSIF tyP0921InletNOutletShutter.tyNaviOutlet21.tyBtnRgt.bRtCompl THEN
		//outlet 2 navi
		p_tyC0004Navi ACCESS ADR (tyP0921InletNOutletShutter.tyNaviOutlet22);
		tyP0921InletNOutletShutter.tyOutletShutterCom2.tyTxtTit.usiValueIdx := 149-6; //6

		tyP0921InletNOutletShutter.tyInletShutterCom.tyLyr.uiRtStat := TRUE;
		tyP0921InletNOutletShutter.tyInletShutterFB.tyLyr.uiRtStat := TRUE;
		tyP0921InletNOutletShutter.tyInletShutterDC.tyLyr.uiRtStat := TRUE;

		p_tyP0921OutletShutterCom ACCESS ADR(tyP0921InletNOutletShutter.tyOutletShutterCom2);
		p_tyP0921OutletShutterDC ACCESS ADR(tyP0921InletNOutletShutter.tyOutletShutterDC2);
		p_tyP0921OutletShutterFB ACCESS ADR(tyP0921InletNOutletShutter.tyOutletShutterFB2);
		p_tyP0921OutletShutterDis ACCESS ADR(tyP0921InletNOutletShutter.tyOutletShutterDis);

//		tyP0921InletNOutletShutter.tyOutletShutterDC2.tyBtnOpen2.uiRtStat := TRUE;
//		tyP0921InletNOutletShutter.tyOutletShutterDC2.tyBtnOpen3.uiRtStat := TRUE;
		tyP0921InletNOutletShutter.tyOutletShutterDis.tyLyr.uiRtStat.0 := TRUE;
		tyP0921InletNOutletShutter.tyNaviOutlet21.tyBtnRgt.bRtCompl := FALSE;
		tyP0921InletNOutletShutter.tyNaviOutlet21.tyBitmapPageDisp.usiValueIdx :=2;
		tyP0921InletNOutletShutter.tyNaviOutlet22.tyBitmapPageDisp.usiValueIdx :=2;

	ELSIF tyP0921InletNOutletShutter.tyNaviOutlet21.tyBtnLeft.bRtCompl THEN
		//outlet 2 navi
		p_tyC0004Navi ACCESS ADR (tyP0921InletNOutletShutter.tyNaviOutlet22);
		tyP0921InletNOutletShutter.tyOutletShutterCom2.tyTxtTit.usiValueIdx := 149-6; //6 //title

		tyP0921InletNOutletShutter.tyInletShutterCom.tyLyr.uiRtStat := TRUE;
		tyP0921InletNOutletShutter.tyInletShutterFB.tyLyr.uiRtStat := TRUE;
		tyP0921InletNOutletShutter.tyInletShutterDC.tyLyr.uiRtStat := TRUE;

		p_tyP0921OutletShutterCom ACCESS ADR(tyP0921InletNOutletShutter.tyOutletShutterCom2);
		p_tyP0921OutletShutterDC ACCESS ADR(tyP0921InletNOutletShutter.tyOutletShutterDC2);
		p_tyP0921OutletShutterFB ACCESS ADR(tyP0921InletNOutletShutter.tyOutletShutterFB2);
		p_tyP0921OutletShutterDis ACCESS ADR(tyP0921InletNOutletShutter.tyOutletShutterDis);

//		tyP0921InletNOutletShutter.tyOutletShutterDC2.tyBtnOpen2.uiRtStat := TRUE;
//		tyP0921InletNOutletShutter.tyOutletShutterDC2.tyBtnOpen3.uiRtStat := TRUE;
		tyP0921InletNOutletShutter.tyOutletShutterDis.tyLyr.uiRtStat.0 := TRUE;
		tyP0921InletNOutletShutter.tyNaviOutlet21.tyBtnLeft.bRtCompl := FALSE;
		tyP0921InletNOutletShutter.tyNaviOutlet21.tyBitmapPageDisp.usiValueIdx :=2;
		tyP0921InletNOutletShutter.tyNaviOutlet22.tyBitmapPageDisp.usiValueIdx :=2;

	END_IF

END_ACTION
```

#### Act_OptP0921DualMask.st
```iecst
ACTION Act_OptP0921DualMask:

	IF eCurrPage = UIP0921Shutter THEN

		IF p_tyDI.bEStopSig = FALSE THEN
			p_tyC0003DualMask ACCESS ADR(tyP0921InletNOutletShutter.tyDualMaskEStop);

			tyP0921InletNOutletShutter.tyDualMaskEStop.tyBtnLeftMask.uiMaskRtStat.0	:= NOT p_tyNtParamCurr.bProjInletShutPrep;
			tyP0921InletNOutletShutter.tyDualMaskEStop.tyBtnRgtMask.uiMaskRtStat.0	:= NOT p_tyNtParamCurr.bProjOutletShutPrep;

		ELSIF p_tyDI.bCoverSWSig = FALSE THEN
			p_tyC0003DualMask ACCESS ADR(tyP0921InletNOutletShutter.tyDualMaskCWSig);

			tyP0921InletNOutletShutter.tyDualMaskCWSig.tyBtnLeftMask.uiMaskRtStat.0	:= NOT p_tyNtParamCurr.bProjInletShutPrep;
			tyP0921InletNOutletShutter.tyDualMaskCWSig.tyBtnRgtMask.uiMaskRtStat.0	:= NOT p_tyNtParamCurr.bProjOutletShutPrep;

		ELSIF p_tyDI.bSafetyRlySig = FALSE THEN
			p_tyC0003DualMask ACCESS ADR(tyP0921InletNOutletShutter.tyDualMaskSafetyRly);

			tyP0921InletNOutletShutter.tyDualMaskSafetyRly.tyBtnLeftMask.uiMaskRtStat.0	:= NOT p_tyNtParamCurr.bProjInletShutPrep;
			tyP0921InletNOutletShutter.tyDualMaskSafetyRly.tyBtnRgtMask.uiMaskRtStat.0	:= NOT p_tyNtParamCurr.bProjOutletShutPrep;

		ELSIF p_eLifterBtmStatus = Busy AND p_bLifterBtmPwrOn THEN
			p_tyC0003DualMask ACCESS ADR(tyP0921InletNOutletShutter.tyDualMaskLifMovInterrupt);

			tyP0921InletNOutletShutter.tyDualMaskLifMovInterrupt.tyBtnLeftMask.uiMaskRtStat.0	:= NOT p_tyNtParamCurr.bProjInletShutPrep;
			tyP0921InletNOutletShutter.tyDualMaskLifMovInterrupt.tyBtnRgtMask.uiMaskRtStat.0	:= NOT p_tyNtParamCurr.bProjOutletShutPrep;

		ELSIF p_eTravStatus = Busy AND p_bTravPwrOn THEN
			p_tyC0003DualMask ACCESS ADR(tyP0921InletNOutletShutter.tyDualMaskTravMovInterrupt);

			tyP0921InletNOutletShutter.tyDualMaskTravMovInterrupt.tyBtnLeftMask.uiMaskRtStat.0	:= NOT p_tyNtParamCurr.bProjInletShutPrep;
			tyP0921InletNOutletShutter.tyDualMaskTravMovInterrupt.tyBtnRgtMask.uiMaskRtStat.0	:= NOT p_tyNtParamCurr.bProjOutletShutPrep;

		ELSIF p_eAWOpenStatus = Busy AND p_bAWOpenPwrOn THEN
			p_tyC0003DualMask ACCESS ADR(tyP0921InletNOutletShutter.tyDualMaskAWMovInterrupt);

			tyP0921InletNOutletShutter.tyDualMaskAWMovInterrupt.tyBtnLeftMask.uiMaskRtStat.0	:= NOT p_tyNtParamCurr.bProjInletShutPrep;
			tyP0921InletNOutletShutter.tyDualMaskAWMovInterrupt.tyBtnRgtMask.uiMaskRtStat.0		:= NOT p_tyNtParamCurr.bProjOutletShutPrep;

		ELSIF p_tyDI.bPullerRetRS = FALSE THEN
			p_tyC0003DualMask ACCESS ADR(tyP0921InletNOutletShutter.tyDualMaskPullInterruptInlet);
			IF tyP0921InletNOutletShutter.tyNaviLyr1.tyBitmapPageDisp.usiValueIdx = 1 AND
				ABS(p_diTravActualPos - p_diMagRcp1TravPos) < 290000 THEN
				tyP0921InletNOutletShutter.tyDualMaskPullInterruptInlet.tyBtnLeftMask.uiMaskRtStat := 0;
				tyP0921InletNOutletShutter.tyDualMaskPullInterruptInlet.tyBtnRgtMask.uiMaskRtStat := 1;
			ELSIF tyP0921InletNOutletShutter.tyNaviLyr2.tyBitmapPageDisp.usiValueIdx = 2 AND
				ABS(p_diTravActualPos - p_diMagRcp2TravPos) < 290000 THEN
				tyP0921InletNOutletShutter.tyDualMaskPullInterruptInlet.tyBtnLeftMask.uiMaskRtStat := 0;
				tyP0921InletNOutletShutter.tyDualMaskPullInterruptInlet.tyBtnRgtMask.uiMaskRtStat := 1;
			ELSIF tyP0921InletNOutletShutter.tyNaviLyr2.tyBitmapPageDisp.usiValueIdx = 2 AND
				ABS(p_diTravActualPos - p_diMagRcp3TravPos) < 290000 THEN
				tyP0921InletNOutletShutter.tyDualMaskPullInterruptInlet.tyBtnLeftMask.uiMaskRtStat := 1;
				tyP0921InletNOutletShutter.tyDualMaskPullInterruptInlet.tyBtnRgtMask.uiMaskRtStat := 0;
			ELSE
				tyP0921InletNOutletShutter.tyDualMaskPullInterruptInlet.tyBtnLeftMask.uiMaskRtStat := 1;
				tyP0921InletNOutletShutter.tyDualMaskPullInterruptInlet.tyBtnRgtMask.uiMaskRtStat := 1;
			END_IF

		ELSE
			p_tyC0003DualMask ACCESS ADR(tyP0921InletNOutletShutter.tyDualMaskHide);

		END_IF

	END_IF

END_ACTION
```

#### Act_OptP0921InletShutterChgLyr.st
```iecst
ACTION Act_OptP0921InletShutterChgLyr:

//	tyP0921InletNOutletShutter.tyInletShutterFB.tyLyr.uiRtStat.0	:= NOT(p_tyNtParamCurr.bProjInletShutPrep);

	IF p_tyNtParamCurr.bProjInletShutPrep THEN
		IF tyP0921InletNOutletShutter.tyInletShutterCom.tyBtnSwitch.bRtCompl THEN
			tyP0921InletNOutletShutter.tyInletShutterCom.tyBtnSwitch.bRtCompl := FALSE;

			IF tyP0921InletNOutletShutter.tyInletShutterCom.tyBtnSwitch.bValue = TRUE THEN
				fUIInRtStatOff(ADR(tyP0921InletNOutletShutter.tyInletShutterDC.tyLyr.uiRtStat));
				fUIInRtStatHide(ADR(tyP0921InletNOutletShutter.tyInletShutterFB.tyLyr.uiRtStat));
			ELSE
				fUIInRtStatHide(ADR(tyP0921InletNOutletShutter.tyInletShutterDC.tyLyr.uiRtStat));
				fUIInRtStatOff(ADR(tyP0921InletNOutletShutter.tyInletShutterFB.tyLyr.uiRtStat));
			END_IF

		END_IF
	ELSE
		fUIInRtStatHide(ADR(tyP0921InletNOutletShutter.tyInletShutterDC.tyLyr.uiRtStat));
		fUIInRtStatHide(ADR(tyP0921InletNOutletShutter.tyInletShutterFB.tyLyr.uiRtStat));

	END_IF

END_ACTION
```

#### Act_OptP0921InletShutterSen.st
```iecst
ACTION Act_OptP0921InletShutterSen:

	tyP0921InletNOutletShutter.tyInletShutterCom.tyBtnOpenRS.bValue		:= p_tyDI.bInShutterOpenRS;
	tyP0921InletNOutletShutter.tyInletShutterCom.tyBtnCloseRS.bValue	:= p_tyDI.bInShutterCloseRS;

	//Machine Bitmap //inlet 13close ,14open ; outlet 15open 16close ;; curtain close
	IF   (p_tyNtParamCurr.eProjMag = LDMagDual AND p_tyNtParamCurr.bMagAutoVerifyPrep = FALSE)
		OR (p_tyNtParamCurr.eProjMag = LDMagTriple AND p_tyNtParamCurr.bMagAutoVerifyPrep = FALSE)
		OR (p_tyNtParamCurr.eProjMag = LDMagDual AND p_tyNtParamCurr.bMagAutoVerifyPrep = TRUE)	THEN
		IF p_tyDI.bInShutterOpenRS = TRUE THEN
			tyP0921InletNOutletShutter.tyInletShutterCom.tyBitmapMc.uiValueIdx	:= 1;
		ELSIF p_tyNtParamCurr.bProjCurtainSenPrep THEN
			tyP0921InletNOutletShutter.tyInletShutterCom.tyBitmapMc.uiValueIdx	:= 0+4; //16
		ELSE
			tyP0921InletNOutletShutter.tyInletShutterCom.tyBitmapMc.uiValueIdx	:= 0;
		END_IF
	ELSIF p_tyNtParamCurr.eProjMag = LDMagTriple AND p_tyNtParamCurr.bMagAutoVerifyPrep = TRUE THEN
		IF p_tyDI.bInShutterOpenRS = TRUE THEN
			tyP0921InletNOutletShutter.tyInletShutterCom.tyBitmapMc.uiValueIdx	:= 28;
		ELSE
			tyP0921InletNOutletShutter.tyInletShutterCom.tyBitmapMc.uiValueIdx	:= 27;
		END_IF

	ELSIF p_tyNtParamCurr.eProjMag = LDMagQuadruple AND p_tyNtParamCurr.bMagAutoVerifyPrep = TRUE THEN
		IF p_tyDI.bInShutterOpenRS = TRUE THEN
			tyP0921InletNOutletShutter.tyInletShutterCom.tyBitmapMc.uiValueIdx	:= 51;
		ELSE
			tyP0921InletNOutletShutter.tyInletShutterCom.tyBitmapMc.uiValueIdx	:= 50;
		END_IF
	END_IF

	//Add
	IF p_tyNtParamCurr.eProjMag = LDMagTriple AND p_tyNtParamCurr.bProjLifterMagPlatform THEN
		IF 	tyP0921InletNOutletShutter.tyInletShutterCom.tyBitmapMc.uiValueIdx < 400 THEN
			tyP0921InletNOutletShutter.tyInletShutterCom.tyBitmapMc.uiValueIdx	:= tyP0921InletNOutletShutter.tyInletShutterCom.tyBitmapMc.uiValueIdx + 400;
		END_IF
	ELSIF p_tyNtParamCurr.eProjMag = LDMagTriple AND p_tyNtParamCurr.bMagAutoVerifyPrep = FALSE AND p_tyNtParamCurr.bProjMotorizedPullerPrep = FALSE THEN
		IF 	tyP0921InletNOutletShutter.tyInletShutterCom.tyBitmapMc.uiValueIdx < 300 THEN //100 cannot use
			tyP0921InletNOutletShutter.tyInletShutterCom.tyBitmapMc.uiValueIdx	:= tyP0921InletNOutletShutter.tyInletShutterCom.tyBitmapMc.uiValueIdx + 300;
		END_IF
	ELSIF p_tyNtParamCurr.eProjMag = LDMagTriple AND p_tyNtParamCurr.bMagAutoVerifyPrep = FALSE AND p_tyNtParamCurr.bProjMotorizedPullerPrep
		AND p_tyNtParamCurr.bProjCurtainSenPrep THEN //curtain
		IF 	tyP0921InletNOutletShutter.tyInletShutterCom.tyBitmapMc.uiValueIdx < 375-14 THEN
			tyP0921InletNOutletShutter.tyInletShutterCom.tyBitmapMc.uiValueIdx	:= tyP0921InletNOutletShutter.tyInletShutterCom.tyBitmapMc.uiValueIdx + 375-14;
		END_IF
	ELSIF (p_tyNtParamCurr.eProjMag = LDMagDual OR p_tyNtParamCurr.eProjMag = LDMagTriple) AND p_tyNtParamCurr.bMagAutoVerifyPrep = TRUE THEN
		IF 	tyP0921InletNOutletShutter.tyInletShutterCom.tyBitmapMc.uiValueIdx < 200 THEN
			tyP0921InletNOutletShutter.tyInletShutterCom.tyBitmapMc.uiValueIdx	:= tyP0921InletNOutletShutter.tyInletShutterCom.tyBitmapMc.uiValueIdx + 200;
		END_IF
	ELSIF (p_tyNtParamCurr.eProjMag = LDMagDual OR p_tyNtParamCurr.eProjMag = LDMagTriple) AND p_tyNtParamCurr.bMagAutoVerifyPrep = FALSE AND  p_tyNtParamCurr.bProjMotorizedPullerPrep = FALSE THEN
		IF 	tyP0921InletNOutletShutter.tyInletShutterCom.tyBitmapMc.uiValueIdx < 200 THEN
			IF p_tyNtParamCurr.bProjLifterMagPlatform THEN
				tyP0921InletNOutletShutter.tyInletShutterCom.tyBitmapMc.uiValueIdx	:= tyP0921InletNOutletShutter.tyInletShutterCom.tyBitmapMc.uiValueIdx + 247;
			ELSE
				IF p_tyNtParamCurr.sJobNo = '2023-0276A01' THEN
					tyP0921InletNOutletShutter.tyInletShutterCom.tyBitmapMc.uiValueIdx	:= tyP0921InletNOutletShutter.tyInletShutterCom.tyBitmapMc.uiValueIdx + 482-13;
				ELSE
					tyP0921InletNOutletShutter.tyInletShutterCom.tyBitmapMc.uiValueIdx	:= tyP0921InletNOutletShutter.tyInletShutterCom.tyBitmapMc.uiValueIdx + 200;
				END_IF
			END_IF
		END_IF
	ELSIF (p_tyNtParamCurr.eProjMag = LDMagDual OR p_tyNtParamCurr.eProjMag = LDMagTriple) AND p_tyNtParamCurr.bMagAutoVerifyPrep = FALSE AND p_tyNtParamCurr.bProjMotorizedPullerPrep = TRUE THEN
		IF 	tyP0921InletNOutletShutter.tyInletShutterCom.tyBitmapMc.uiValueIdx < 300 THEN
			IF p_tyNtParamCurr.sJobNo = '2023-0258A01' THEN
				tyP0921InletNOutletShutter.tyInletShutterCom.tyBitmapMc.uiValueIdx	:= tyP0921InletNOutletShutter.tyInletShutterCom.tyBitmapMc.uiValueIdx + 452-13;
			ELSE
				tyP0921InletNOutletShutter.tyInletShutterCom.tyBitmapMc.uiValueIdx	:= tyP0921InletNOutletShutter.tyInletShutterCom.tyBitmapMc.uiValueIdx + 300;
			END_IF
		END_IF
	END_IF

END_ACTION
```

#### Act_OptP0921InletShutterFB.st
```iecst
ACTION Act_OptP0921InletShutterFB:

	IF tyP0921InletNOutletShutter.tyInletShutterCom.tyBtnSwitch.bValue = FALSE THEN

		IF tyP0921InletNOutletShutter.tyInletShutterFB.tyBtnOpen.bRtCompl = TRUE THEN
			tyP0921InletNOutletShutter.tyInletShutterFB.tyBtnOpen.bRtCompl	:= FALSE;

			tyP0921InletNOutletShutter.tyInletShutterFB.tyBtnOpen.bValue	:= TRUE;
			tyP0921InletNOutletShutter.tyInletShutterFB.tyBtnClose.bValue	:= FALSE;

		ELSIF tyP0921InletNOutletShutter.tyInletShutterFB.tyBtnClose.bRtCompl = TRUE THEN
			tyP0921InletNOutletShutter.tyInletShutterFB.tyBtnClose.bRtCompl	:= FALSE;

			tyP0921InletNOutletShutter.tyInletShutterFB.tyBtnClose.bValue	:= TRUE;
			tyP0921InletNOutletShutter.tyInletShutterFB.tyBtnOpen.bValue	:= FALSE;
		END_IF

		IF tyP0921InletNOutletShutter.tyInletShutterFB.tyBtnOpen.bValue = TRUE THEN
			eInShutterAct	:= PneuActRet;

			IF p_eInShutterStat = PneuActRet AND p_eInShutterStatus = Done THEN
				eInShutterAct	:= PneuActIdle;

				tyP0921InletNOutletShutter.tyInletShutterFB.tyBtnOpen.bValue	:= FALSE;
			ELSIF p_eInShutterStatus = Error THEN
				tyP0921InletNOutletShutter.tyInletShutterFB.tyBtnOpen.bValue	:= FALSE;
			END_IF

		ELSIF tyP0921InletNOutletShutter.tyInletShutterFB.tyBtnClose.bValue = TRUE THEN
			eInShutterAct	:= PneuActExt;

			IF p_eInShutterStat = PneuActExt AND p_eInShutterStatus = Done THEN
				eInShutterAct	:= PneuActIdle;

				tyP0921InletNOutletShutter.tyInletShutterFB.tyBtnClose.bValue := FALSE;
			ELSIF p_eInShutterStatus = Error THEN
				tyP0921InletNOutletShutter.tyInletShutterFB.tyBtnClose.bValue := FALSE;
			END_IF
		END_IF

		//Update Direct Control Status
		tyP0921InletNOutletShutter.tyInletShutterDC.tyBtnOpen.bRtCompl	:= FALSE;
		tyP0921InletNOutletShutter.tyInletShutterDC.tyBtnClose.bRtCompl	:= FALSE;
		tyP0921InletNOutletShutter.tyInletShutterDC.tyBtnOpen.bValue	:= p_bInShutterRetCtrl;
		tyP0921InletNOutletShutter.tyInletShutterDC.tyBtnClose.bValue	:= p_bInShutterExtCtrl;

	END_IF

END_ACTION
```

#### Act_OptP0921InletShutterDC.st
```iecst
ACTION Act_OptP0921InletShutterDC:

	IF tyP0921InletNOutletShutter.tyInletShutterCom.tyBtnSwitch.bValue = TRUE THEN
		IF p_bInShutterTwoCtrlOut = FALSE THEN
			IF tyP0921InletNOutletShutter.tyInletShutterDC.tyBtnOpen.bRtCompl = TRUE THEN
				tyP0921InletNOutletShutter.tyInletShutterDC.tyBtnOpen.bValue	:= TRUE;
				tyP0921InletNOutletShutter.tyInletShutterDC.tyBtnClose.bValue	:= FALSE;

				eInShutterAct	:= PneuActSetRet;

				IF p_eInShutterStat = PneuActSetRet AND p_eInShutterStatus = Done THEN
					eInShutterAct	:= PneuActIdle;

					tyP0921InletNOutletShutter.tyInletShutterDC.tyBtnOpen.bRtCompl	:= FALSE;
				END_IF

			ELSIF tyP0921InletNOutletShutter.tyInletShutterDC.tyBtnClose.bRtCompl = TRUE THEN
				tyP0921InletNOutletShutter.tyInletShutterDC.tyBtnClose.bValue	:= TRUE;
				tyP0921InletNOutletShutter.tyInletShutterDC.tyBtnOpen.bValue	:= FALSE;

				eInShutterAct	:= PneuActSetExt;

				IF p_eInShutterStat = PneuActSetExt AND p_eInShutterStatus = Done THEN
					eInShutterAct	:= PneuActIdle;

					tyP0921InletNOutletShutter.tyInletShutterDC.tyBtnClose.bRtCompl	:= FALSE;
				END_IF
			END_IF

		ELSE
			IF (tyP0921InletNOutletShutter.tyInletShutterDC.tyBtnOpen.bRtCompl = TRUE) OR (tyP0921InletNOutletShutter.tyInletShutterDC.tyBtnClose.bRtCompl = TRUE) THEN
				IF (tyP0921InletNOutletShutter.tyInletShutterDC.tyBtnOpen.bValue = TRUE) AND (tyP0921InletNOutletShutter.tyInletShutterDC.tyBtnClose.bValue = TRUE) THEN
					eInShutterAct	:= PneuActSetAll;

					IF p_eInShutterStat = PneuActSetAll AND p_eInShutterStatus = Done THEN
						eInShutterAct	:= PneuActIdle;

						tyP0921InletNOutletShutter.tyInletShutterDC.tyBtnOpen.bRtCompl	:= FALSE;
						tyP0921InletNOutletShutter.tyInletShutterDC.tyBtnClose.bRtCompl	:= FALSE;
					END_IF

				ELSIF (tyP0921InletNOutletShutter.tyInletShutterDC.tyBtnOpen.bValue = TRUE) AND (tyP0921InletNOutletShutter.tyInletShutterDC.tyBtnClose.bValue = FALSE) THEN
					eInShutterAct	:= PneuActSetRet;

					IF p_eInShutterStat = PneuActSetRet AND p_eInShutterStatus = Done THEN
						eInShutterAct	:= PneuActIdle;

						tyP0921InletNOutletShutter.tyInletShutterDC.tyBtnOpen.bRtCompl	:= FALSE;
						tyP0921InletNOutletShutter.tyInletShutterDC.tyBtnClose.bRtCompl	:= FALSE;
					END_IF

				ELSIF (tyP0921InletNOutletShutter.tyInletShutterDC.tyBtnOpen.bValue = FALSE) AND (tyP0921InletNOutletShutter.tyInletShutterDC.tyBtnClose.bValue = TRUE) THEN
					eInShutterAct	:= PneuActSetExt;

					IF p_eInShutterStat = PneuActSetExt AND p_eInShutterStatus = Done THEN
						eInShutterAct	:= PneuActIdle;

						tyP0921InletNOutletShutter.tyInletShutterDC.tyBtnOpen.bRtCompl	:= FALSE;
						tyP0921InletNOutletShutter.tyInletShutterDC.tyBtnClose.bRtCompl	:= FALSE;
					END_IF

				ELSE
					eInShutterAct	:= PneuActRstAll;

					IF p_eInShutterStat = PneuActRstAll AND p_eInShutterStatus = Done THEN
						eInShutterAct	:= PneuActIdle;

						tyP0921InletNOutletShutter.tyInletShutterDC.tyBtnOpen.bRtCompl	:= FALSE;
						tyP0921InletNOutletShutter.tyInletShutterDC.tyBtnClose.bRtCompl	:= FALSE;
					END_IF

				END_IF
			END_IF
		END_IF

		tyP0921InletNOutletShutter.tyInletShutterFB.tyBtnClose.bRtCompl	:= FALSE;
		tyP0921InletNOutletShutter.tyInletShutterFB.tyBtnClose.bValue	:= FALSE;
		tyP0921InletNOutletShutter.tyInletShutterFB.tyBtnOpen.bRtCompl	:= FALSE;
		tyP0921InletNOutletShutter.tyInletShutterFB.tyBtnOpen.bValue	:= FALSE;

	END_IF

END_ACTION
```

#### Act_OptP0921OutletShutterChgLyr.st
```iecst
ACTION Act_OptP0921OutletShutterChgLyr:

//	tyP0921InletNOutletShutter.tyOutletShutterFB.tyLyr.uiRtStat.0	:= NOT(p_tyNtParamCurr.bProjOutletShutPrep);

	IF p_tyNtParamCurr.bProjOutletShutPrep THEN
		IF	tyP0921InletNOutletShutter.tyOutletShutterCom.tyBtnSwitch.bRtCompl THEN
				tyP0921InletNOutletShutter.tyOutletShutterCom.tyBtnSwitch.bRtCompl := FALSE;

			IF tyP0921InletNOutletShutter.tyOutletShutterCom.tyBtnSwitch.bValue = TRUE THEN
				fUIInRtStatOff(ADR(tyP0921InletNOutletShutter.tyOutletShutterDC.tyLyr.uiRtStat));
				fUIInRtStatHide(ADR(tyP0921InletNOutletShutter.tyOutletShutterFB.tyLyr.uiRtStat));
			ELSE
				fUIInRtStatHide(ADR(tyP0921InletNOutletShutter.tyOutletShutterDC.tyLyr.uiRtStat));
				fUIInRtStatOff(ADR(tyP0921InletNOutletShutter.tyOutletShutterFB.tyLyr.uiRtStat));
			END_IF

		END_IF
	ELSE
		fUIInRtStatHide(ADR(tyP0921InletNOutletShutter.tyOutletShutterDC.tyLyr.uiRtStat));
		fUIInRtStatHide(ADR(tyP0921InletNOutletShutter.tyOutletShutterFB.tyLyr.uiRtStat));

	END_IF

END_ACTION
```

#### Act_OptP0921OutletShutterSen.st
```iecst
ACTION Act_OptP0921OutletShutterSen:

	tyP0921InletNOutletShutter.tyOutletShutterCom.tyBtnOpenRS.bValue	:= p_tyDI.bOutShutterOpenRS;
	tyP0921InletNOutletShutter.tyOutletShutterCom.tyBtnCloseRS.bValue	:= p_tyDI.bOutShutterCloseRS;

	//Machine Bitmap //15open ,16close
	IF   (p_tyNtParamCurr.eProjMag = LDMagDual AND p_tyNtParamCurr.bMagAutoVerifyPrep = FALSE)
		OR (p_tyNtParamCurr.eProjMag = LDMagTriple AND p_tyNtParamCurr.bMagAutoVerifyPrep = FALSE)
		OR (p_tyNtParamCurr.eProjMag = LDMagDual AND p_tyNtParamCurr.bMagAutoVerifyPrep = TRUE)
		THEN
		IF p_tyDI.bOutShutterOpenRS = TRUE THEN
			tyP0921InletNOutletShutter.tyOutletShutterCom.tyBitmapMc.uiValueIdx	:= 1;
		ELSE
			tyP0921InletNOutletShutter.tyOutletShutterCom.tyBitmapMc.uiValueIdx	:= 0;
		END_IF
	ELSIF p_tyNtParamCurr.eProjMag = LDMagTriple AND p_tyNtParamCurr.bMagAutoVerifyPrep = TRUE
		THEN
		IF p_tyDI.bOutShutterOpenRS = TRUE THEN
			tyP0921InletNOutletShutter.tyOutletShutterCom.tyBitmapMc.uiValueIdx	:= 28;
		ELSE
			tyP0921InletNOutletShutter.tyOutletShutterCom.tyBitmapMc.uiValueIdx	:= 27;
		END_IF
	ELSIF p_tyNtParamCurr.eProjMag = LDMagQuadruple AND p_tyNtParamCurr.bMagAutoVerifyPrep = TRUE
		THEN
		IF p_tyDI.bOutShutterOpenRS = TRUE THEN
			tyP0921InletNOutletShutter.tyOutletShutterCom.tyBitmapMc.uiValueIdx	:= 51;
		ELSE
			tyP0921InletNOutletShutter.tyOutletShutterCom.tyBitmapMc.uiValueIdx	:= 50;
		END_IF
	END_IF

	IF p_tyNtParamCurr.eProjMag = LDMagTriple AND p_tyNtParamCurr.bProjLifterMagPlatform THEN //same with bosch curtain
		IF 	tyP0921InletNOutletShutter.tyOutletShutterCom.tyBitmapMc.uiValueIdx < 400 THEN
			tyP0921InletNOutletShutter.tyOutletShutterCom.tyBitmapMc.uiValueIdx	:= tyP0921InletNOutletShutter.tyOutletShutterCom.tyBitmapMc.uiValueIdx + 400;
		END_IF
	ELSIF p_tyNtParamCurr.eProjMag = LDMagTriple AND p_tyNtParamCurr.bMagAutoVerifyPrep = FALSE AND p_tyNtParamCurr.bProjMotorizedPullerPrep = FALSE
		THEN
		IF 	tyP0921InletNOutletShutter.tyOutletShutterCom.tyBitmapMc.uiValueIdx < 100 THEN
			tyP0921InletNOutletShutter.tyOutletShutterCom.tyBitmapMc.uiValueIdx	:= tyP0921InletNOutletShutter.tyOutletShutterCom.tyBitmapMc.uiValueIdx + 100;
		END_IF
	ELSIF p_tyNtParamCurr.eProjMag = LDMagTriple AND p_tyNtParamCurr.bMagAutoVerifyPrep = FALSE AND p_tyNtParamCurr.bProjMotorizedPullerPrep = TRUE
		AND p_tyNtParamCurr.bProjCurtainSenPrep THEN //curtain
		IF 	tyP0921InletNOutletShutter.tyOutletShutterCom.tyBitmapMc.uiValueIdx < 387-15 THEN
			tyP0921InletNOutletShutter.tyOutletShutterCom.tyBitmapMc.uiValueIdx	:= tyP0921InletNOutletShutter.tyOutletShutterCom.tyBitmapMc.uiValueIdx + 387-15;
		END_IF
	ELSIF (p_tyNtParamCurr.eProjMag = LDMagDual OR p_tyNtParamCurr.eProjMag = LDMagTriple)
		AND p_tyNtParamCurr.bMagAutoVerifyPrep = TRUE
		THEN
		IF 	tyP0921InletNOutletShutter.tyOutletShutterCom.tyBitmapMc.uiValueIdx < 200 THEN
			tyP0921InletNOutletShutter.tyOutletShutterCom.tyBitmapMc.uiValueIdx	:= tyP0921InletNOutletShutter.tyOutletShutterCom.tyBitmapMc.uiValueIdx + 200;
		END_IF
	ELSIF (p_tyNtParamCurr.eProjMag = LDMagDual OR p_tyNtParamCurr.eProjMag = LDMagTriple)
		AND p_tyNtParamCurr.bMagAutoVerifyPrep = FALSE  AND p_tyNtParamCurr.bProjMotorizedPullerPrep = TRUE
		THEN
		IF 	tyP0921InletNOutletShutter.tyOutletShutterCom.tyBitmapMc.uiValueIdx < 300 THEN
			IF p_tyNtParamCurr.sJobNo = '2023-0258A01' THEN
				tyP0921InletNOutletShutter.tyOutletShutterCom.tyBitmapMc.uiValueIdx	:= tyP0921InletNOutletShutter.tyOutletShutterCom.tyBitmapMc.uiValueIdx + 454-15;
			ELSE
				tyP0921InletNOutletShutter.tyOutletShutterCom.tyBitmapMc.uiValueIdx	:= tyP0921InletNOutletShutter.tyOutletShutterCom.tyBitmapMc.uiValueIdx + 300;
			END_IF
		END_IF
	ELSIF (p_tyNtParamCurr.eProjMag = LDMagDual OR p_tyNtParamCurr.eProjMag = LDMagTriple)
		AND p_tyNtParamCurr.bMagAutoVerifyPrep = FALSE  AND p_tyNtParamCurr.bProjMotorizedPullerPrep = FALSE
		THEN
		IF 	tyP0921InletNOutletShutter.tyOutletShutterCom.tyBitmapMc.uiValueIdx < 200 THEN
			IF p_tyNtParamCurr.bProjLifterMagPlatform THEN
				tyP0921InletNOutletShutter.tyOutletShutterCom.tyBitmapMc.uiValueIdx	:= tyP0921InletNOutletShutter.tyOutletShutterCom.tyBitmapMc.uiValueIdx + 247;
			ELSE
				IF p_tyNtParamCurr.sJobNo = '2023-0276A01' THEN
					tyP0921InletNOutletShutter.tyOutletShutterCom.tyBitmapMc.uiValueIdx	:= tyP0921InletNOutletShutter.tyOutletShutterCom.tyBitmapMc.uiValueIdx + 484-15;
				ELSE
					tyP0921InletNOutletShutter.tyOutletShutterCom.tyBitmapMc.uiValueIdx	:= tyP0921InletNOutletShutter.tyOutletShutterCom.tyBitmapMc.uiValueIdx + 200;
				END_IF
			END_IF
		END_IF
	END_IF
	END_ACTION
```

#### Act_OptP0921OutletShutterFB.st
```iecst
ACTION Act_OptP0921OutletShutterFB:

	IF tyP0921InletNOutletShutter.tyOutletShutterCom.tyBtnSwitch.bValue = FALSE THEN
		// FB Control
		IF tyP0921InletNOutletShutter.tyOutletShutterFB.tyBtnOpen.bRtCompl = TRUE THEN
			tyP0921InletNOutletShutter.tyOutletShutterFB.tyBtnOpen.bRtCompl	:= FALSE;

			tyP0921InletNOutletShutter.tyOutletShutterFB.tyBtnOpen.bValue	:= TRUE;
			tyP0921InletNOutletShutter.tyOutletShutterFB.tyBtnClose.bValue	:= FALSE;

		ELSIF tyP0921InletNOutletShutter.tyOutletShutterFB.tyBtnClose.bRtCompl = TRUE THEN
			tyP0921InletNOutletShutter.tyOutletShutterFB.tyBtnClose.bRtCompl	:= FALSE;

			tyP0921InletNOutletShutter.tyOutletShutterFB.tyBtnClose.bValue	:= TRUE;
			tyP0921InletNOutletShutter.tyOutletShutterFB.tyBtnOpen.bValue	:= FALSE;
		END_IF

		IF tyP0921InletNOutletShutter.tyOutletShutterFB.tyBtnOpen.bValue = TRUE THEN
			eOutShutterAct	:= PneuActRet;

			IF p_eOutShutterStat = PneuActRet AND p_eOutShutterStatus = Done THEN
				eOutShutterAct	:= PneuActIdle;

				tyP0921InletNOutletShutter.tyOutletShutterFB.tyBtnOpen.bValue	:= FALSE;
			ELSIF p_eOutShutterStatus = Error THEN
				tyP0921InletNOutletShutter.tyOutletShutterFB.tyBtnOpen.bValue	:= FALSE;
			END_IF

		ELSIF tyP0921InletNOutletShutter.tyOutletShutterFB.tyBtnClose.bValue = TRUE THEN
			eOutShutterAct	:= PneuActExt;

			IF p_eOutShutterStat = PneuActExt AND p_eOutShutterStatus = Done THEN
				eOutShutterAct	:= PneuActIdle;

				tyP0921InletNOutletShutter.tyOutletShutterFB.tyBtnClose.bValue := FALSE;
			ELSIF p_eOutShutterStatus = Error THEN
				tyP0921InletNOutletShutter.tyOutletShutterFB.tyBtnClose.bValue := FALSE;
			END_IF
		END_IF

		//UpdateStatus
		tyP0921InletNOutletShutter.tyOutletShutterDC.tyBtnClose.bRtCompl	:= FALSE;
		tyP0921InletNOutletShutter.tyOutletShutterDC.tyBtnOpen.bRtCompl		:= FALSE;
		tyP0921InletNOutletShutter.tyOutletShutterDC.tyBtnClose.bValue		:= p_bOutShutterExtCtrl;
		tyP0921InletNOutletShutter.tyOutletShutterDC.tyBtnOpen.bValue		:= p_bOutShutterRetCtrl;

	END_IF

END_ACTION
```
